// TIA Portal V20 export
// export: Created 2025-12-01T14:57:40.1723845Z, ExportSetting None, DisplayName Totally Integrated Automation Portal, DisplayVersion V20 Update 3, DisplayName TIA Portal Openness, DisplayVersion V20 Update 3, DisplayName TIA Portal Version Control Interface, DisplayVersion V20 Update 3, DisplayName STEP 7 Professional, DisplayVersion V20 Update 3, DisplayName STEP 7 Safety, DisplayVersion V20 Update 2, DisplayName WinCC Basic/Comfort/Advanced, DisplayVersion V20 Update 3, DisplayName WinCC Professional, DisplayVersion V20 Update 3, DisplayName WinCC Unified, DisplayVersion V20 Update 3
FUNCTION_BLOCK "FB159_M_PASO_E0E3_S0S3_RechazoFruta"   // FB159, LAD
TITLE = Control del Ramal de Salidas
{ S7_Optimized_Access := 'FALSE' }
AUTHOR : PASO
NAME : 20160509
VERSION : 3.3
// stored: AutoNumber false, SetENOAutomatically false
   VAR_INPUT
      Mesa : UInt;   // Mesa de la FB
      Error_Tx : Bool;   // Error en el Tx
      EnTension : Bool;   // Existe Tension en la Mesa
      Termico_Tx : Bool;   // Proteccion del Tx
      pHsMx_Carretilla : Bool;   // pHs de Carretilla
      pHsMx : Bool;   // pHs de la Mesa
      pHsMx_PR3 : Bool;   // pHs de Protrusion de la Mesa. Nota: No existe >> ON
      EnMovimiento_Tx : Bool;   // Avance o Retroceso del Tx
      MAnt_DescargaAct : Bool;   // E1 >> Mesa Anterior DescargaAct
      AVTF_MAnt_Mx : Bool;   // E1 >> Mesa Anterior AVTF
      P_Mens_MAnt_Mx : Bool;   // E1 >> Mesa Anterior P_Mens
      PTF_Mx_MSig : Bool;   // S3 >> Mesa Siguiente PTF
      FTF_Mx_MSig : Bool;   // S3 >> Mesa Siguiente FTF
      MSig_CargaAct : Bool;
      Mx_Centraje : Bool;   // Config >> Activar Centraje de Carga
      Mx_VelocidadLenta_In : Bool;   // Forzar a Velociada Lenta
      F_ENV_MENS_Mx : Bool;   // Fin de Envio de Mensaje
      OrdSal_S03 : Bool;   // Orden de Salida por S3
      OrdSal_S00 : Bool;   // Orden de Salida por S0
      V_CNT_pHsMx : Int := 1000;   // Valor de Presencia
      V_CNT_pHsMx_FTF : Int := 200;   // Valor para activar FTF. Nota: < = V_CNT_pHsMx.
      V_CNTSeg_pHsMx : Int := 2000;   // Valor de Seguriadad para Presencia
      V_CNT_PasoLenta : Int := 2000;   // Valor de Paso a Lenta
      V_CNT_AphsMx : Int := 500;   // Valor de Ausencia
      V_CNTSeg_ApHsMx : Int := 2000;   // Valor de Seguriadad para Ausencia
      V_TMP_Entrada : Int := 5000;   // Valor de Entrada de Carga >> E0
      V_TMP_Retirar : Int := 5000;   // Valor de Retirada de Carga >> S0
      V_CNT_Centrado : Int := 2000;   // Valor de Centrado de Carga
      V_CNT_Reposo : Int := 3000;   // Valor de Reposo de Carga Nota: > Centrado
      V_TOut_Tx_Mx : Int := 15000;   // TimeOut de Entrada por E1
      V_TMP_Protrusion : Int := 200;   // TMP de Protrusion
      V_CNT_PerdidapHs : Int := 1000;   // CNT de Perdida de pHs
   END_VAR
   VAR_OUTPUT
      P_EnvMens_PMx : Bool;   // Permiso de Enviar Mensaje de Presencia
      P_EnvMens_AMx : Bool;   // Permiso de Enviar Mensaje de Ausencia
      P_RecepOK_Mx : Bool;   // Recepcion OK
      PTF_MAnt_Mx : Bool;   // E1 >> Mesa Anterior PTF
      FTF_MAnt_Mx : Bool;   // E1 >> Mesa Anterior FTF
      AVTF_Mx_MSig : Bool;   // S3 >> Mesa Siguiente AVTF
      P_Mens_Mx_MSig : Bool;   // S3 >> Mesa Siguiente P_Mens
   END_VAR
   VAR
      Anular_prE1 : Bool;   // ???
      Anular_prS3 : Bool;   // ???
      Mx_ET00 : Bool;
      Mx_ET01 : Bool;
      Mx_ET02 : Bool;
      Mx_ET08 : Bool;
      Mx_ET09 : Bool;
      Mx_ET10 : Bool;
      Mx_ET11 : Bool;
      Mx_ET12 : Bool;
      Mx_ET110 : Bool;
      Mx_ET111 : Bool;
      Mx_ET40 : Bool;
      Mx_ET41 : Bool;
      Mx_ET42 : Bool;
      Mx_ET43 : Bool;
      Mx_ET140 : Bool;
      Mx_ET141 : Bool;
      Mx_ET50 : Bool;
      Mx_ET51 : Bool;
      Mx_ET150 : Bool;
      Mx_ET151 : Bool;
      Mx_ET90 : Bool;
      Mx_ET91 : Bool;
      Mx_ET190 : Bool;
      Mx_ET191 : Bool;
      Mx_ET192 : Bool;
      ProtocoloIniciado : Bool;   // Iniciado el Envio del Mensaje de Presencia
      CNT_pHsMx_FTF_OK : Bool;   // Enviar ya FTF
      CNT_pHsMx { S7_SetPoint := 'True'} : "FB910_CNT_UHS";   // CNT de la Presencia
      CNTSeg_pHsMx { S7_SetPoint := 'True'} : "FB910_CNT_UHS";   // CNT de Seguridad de la Presencia
      CNT_ApHsMx { S7_SetPoint := 'True'} : "FB910_CNT_UHS";   // CNT de la Ausencia
      CNTSeg_ApHsMx { S7_SetPoint := 'True'} : "FB910_CNT_UHS";   // CNT de Seguridad de la Ausencia
      TMP_Entrada { S7_SetPoint := 'True'} : "FB910_CNT_UHS";   // TMP de Entrada de Carga
      TMP_Retirar { S7_SetPoint := 'True'} : "FB910_CNT_UHS";   // TMP de Retirada de Carga
      CNT_Centrado { S7_SetPoint := 'True'} : "FB910_CNT_UHS";   // Contador de Centrado de Carga
      TMP_EnTension { S7_SetPoint := 'True'} : "FB910_CNT_UHS";
      TOut_Av_Mx { S7_SetPoint := 'True'} : "FB910_CNT_UHS";   // Time Out de Entrada de E1
      TMP_Protrusion { S7_SetPoint := 'True'} : "FB910_CNT_UHS";   // TMP de la Protrusion
      CNT_PerdidapHs { S7_SetPoint := 'True'} : "FB910_CNT_UHS";   // CNT de Perdida de pHs
      STAT_EnvMens_PMx : Bool;   // Interna >> Envio del Mensaje de Presencia
      STAT_EnvMens_AMx : Bool;   // Interna >> Envio de Mensaje de Ausencia
      STAT_FTF_MAnt_Mx : Bool;   // Interna >> FTF de MAnt >> Mx
      STAT_AVTF_Mx_MSig : Bool;   // Interna >> AVTF de Mx >> MSig
      MA_BalizaEntrada : Bool;   // ????
   END_VAR
   VAR_TEMP
      EstadoZona : "EstadoZona";   // Estado de Zona de la Mesa
      EstadoVI : "EstadosMesa";   // Estado del Vehiculo Inteliguente de la Mesa
      ConfigFB : "UDT_ConfigFB";   // Configuracion de la FB de la Mesa
      V_Protrusion : Int;
      Aux_ET00 : Bool;
   END_VAR
BEGIN

REGION Network 1: INICIALIZAR - Recoger las Variables de Estado de la Mesa
   // Se recoge - Estado_CBx
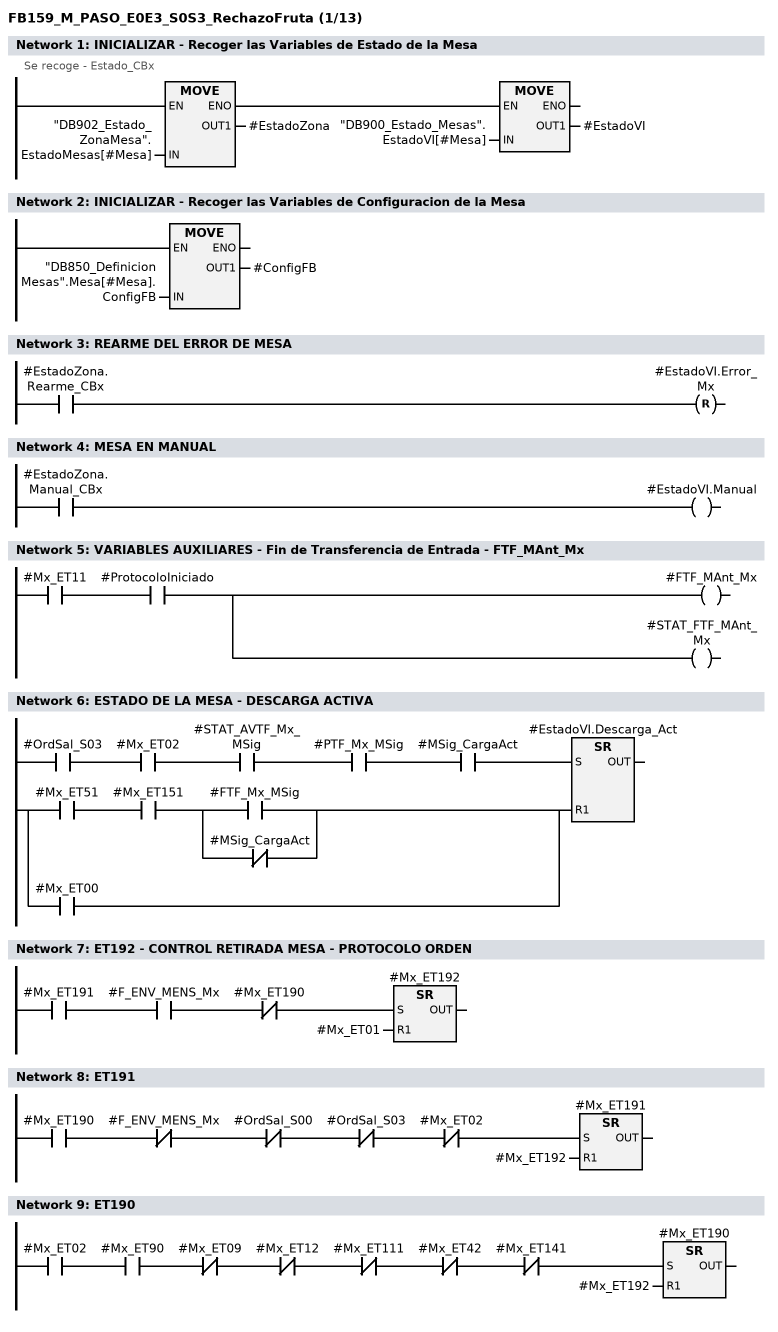
   RUNG wire#powerrail
      Move(in := "DB902_Estado_ZonaMesa".EstadoMesas[#Mesa], out1 => #EstadoZona)
      Move(in := "DB900_Estado_Mesas".EstadoVI[#Mesa], out1 => #EstadoVI)
   END_RUNG
   // the same network as SCL:
   #EstadoZona := "DB902_Estado_ZonaMesa".EstadoMesas[#Mesa];
   #EstadoVI := "DB900_Estado_Mesas".EstadoVI[#Mesa];
END_REGION

REGION Network 2: INICIALIZAR - Recoger las Variables de Configuracion de la Mesa
   RUNG wire#powerrail
      Move(in := "DB850_DefinicionMesas".Mesa[#Mesa].ConfigFB, out1 => #ConfigFB)
   END_RUNG
   // the same network as SCL:
   #ConfigFB := "DB850_DefinicionMesas".Mesa[#Mesa].ConfigFB;
END_REGION

REGION Network 3: REARME DEL ERROR DE MESA
   RUNG wire#powerrail
      Contact( #EstadoZona.Rearme_CBx )
      R_Coil( #EstadoVI.Error_Mx )
   END_RUNG
   // the same network as SCL:
   IF #EstadoZona.Rearme_CBx THEN #EstadoVI.Error_Mx := FALSE; END_IF;
END_REGION

REGION Network 4: MESA EN MANUAL
   RUNG wire#powerrail
      Contact( #EstadoZona.Manual_CBx )
      Coil( #EstadoVI.Manual )
   END_RUNG
   // the same network as SCL:
   #EstadoVI.Manual := #EstadoZona.Manual_CBx;
END_REGION

REGION Network 5: VARIABLES AUXILIARES - Fin de Transferencia de Entrada - FTF_MAnt_Mx
   RUNG wire#powerrail
      Contact( #Mx_ET11 )
      Contact( #ProtocoloIniciado )
      wire#w1
      Coil( #FTF_MAnt_Mx )
   END_RUNG
   RUNG wire#w1
      Coil( #STAT_FTF_MAnt_Mx )
   END_RUNG
   // the same network as SCL:
   #FTF_MAnt_Mx := #Mx_ET11 AND #ProtocoloIniciado;
   #STAT_FTF_MAnt_Mx := #FTF_MAnt_Mx;
END_REGION

REGION Network 6: ESTADO DE LA MESA - DESCARGA ACTIVA
   RUNG wire#powerrail
      Contact( #OrdSal_S03 )
      Contact( #Mx_ET02 )
      Contact( #STAT_AVTF_Mx_MSig )
      Contact( #PTF_Mx_MSig )
      Contact( #MSig_CargaAct )
      S_SR(operand := #EstadoVI.Descarga_Act, r1 := wire#w2)
   END_RUNG
   RUNG wire#powerrail
      Contact( #Mx_ET51 )
      Contact( #Mx_ET151 )
      wire#w1
      Contact( #FTF_Mx_MSig )
   END_RUNG wire#w2
   RUNG wire#w1
      I_Contact( #MSig_CargaAct )
   END_RUNG wire#w2
   RUNG wire#powerrail
      Contact( #Mx_ET00 )
   END_RUNG wire#w2
   // the same network as SCL:
   IF #OrdSal_S03 AND #Mx_ET02 AND #STAT_AVTF_Mx_MSig AND #PTF_Mx_MSig AND #MSig_CargaAct THEN
       #EstadoVI.Descarga_Act := TRUE;   // SR flip-flop
   END_IF;
   IF (#Mx_ET51 AND #Mx_ET151 AND (#FTF_Mx_MSig OR NOT #MSig_CargaAct)) OR #Mx_ET00 THEN
       #EstadoVI.Descarga_Act := FALSE;
   END_IF;
END_REGION

REGION Network 7: ET192 - CONTROL RETIRADA MESA - PROTOCOLO ORDEN
   RUNG wire#powerrail
      Contact( #Mx_ET191 )
      Contact( #F_ENV_MENS_Mx )
      I_Contact( #Mx_ET190 )
      S_SR(operand := #Mx_ET192, r1 := #Mx_ET01)
   END_RUNG
   // the same network as SCL:
   IF #Mx_ET191 AND #F_ENV_MENS_Mx AND NOT #Mx_ET190 THEN
       #Mx_ET192 := TRUE;   // SR flip-flop
   END_IF;
   IF #Mx_ET01 THEN #Mx_ET192 := FALSE; END_IF;
END_REGION

REGION Network 8: ET191
   RUNG wire#powerrail
      Contact( #Mx_ET190 )
      I_Contact( #F_ENV_MENS_Mx )
      I_Contact( #OrdSal_S00 )
      I_Contact( #OrdSal_S03 )
      I_Contact( #Mx_ET02 )
      S_SR(operand := #Mx_ET191, r1 := #Mx_ET192)
   END_RUNG
   // the same network as SCL:
   IF #Mx_ET190 AND NOT #F_ENV_MENS_Mx AND NOT #OrdSal_S00 AND NOT #OrdSal_S03 AND NOT #Mx_ET02 THEN
       #Mx_ET191 := TRUE;   // SR flip-flop
   END_IF;
   IF #Mx_ET192 THEN #Mx_ET191 := FALSE; END_IF;
END_REGION

REGION Network 9: ET190
   RUNG wire#powerrail
      Contact( #Mx_ET02 )
      Contact( #Mx_ET90 )
      I_Contact( #Mx_ET09 )
      I_Contact( #Mx_ET12 )
      I_Contact( #Mx_ET111 )
      I_Contact( #Mx_ET42 )
      I_Contact( #Mx_ET141 )
      S_SR(operand := #Mx_ET190, r1 := #Mx_ET192)
   END_RUNG
   // the same network as SCL:
   IF #Mx_ET02 AND #Mx_ET90 AND NOT #Mx_ET09 AND NOT #Mx_ET12 AND NOT #Mx_ET111 AND NOT #Mx_ET42 AND NOT #Mx_ET141 THEN
       #Mx_ET190 := TRUE;   // SR flip-flop
   END_IF;
   IF #Mx_ET192 THEN #Mx_ET190 := FALSE; END_IF;
END_REGION

REGION Network 10: ET91 - CONTROL RETIRAR DE MESA
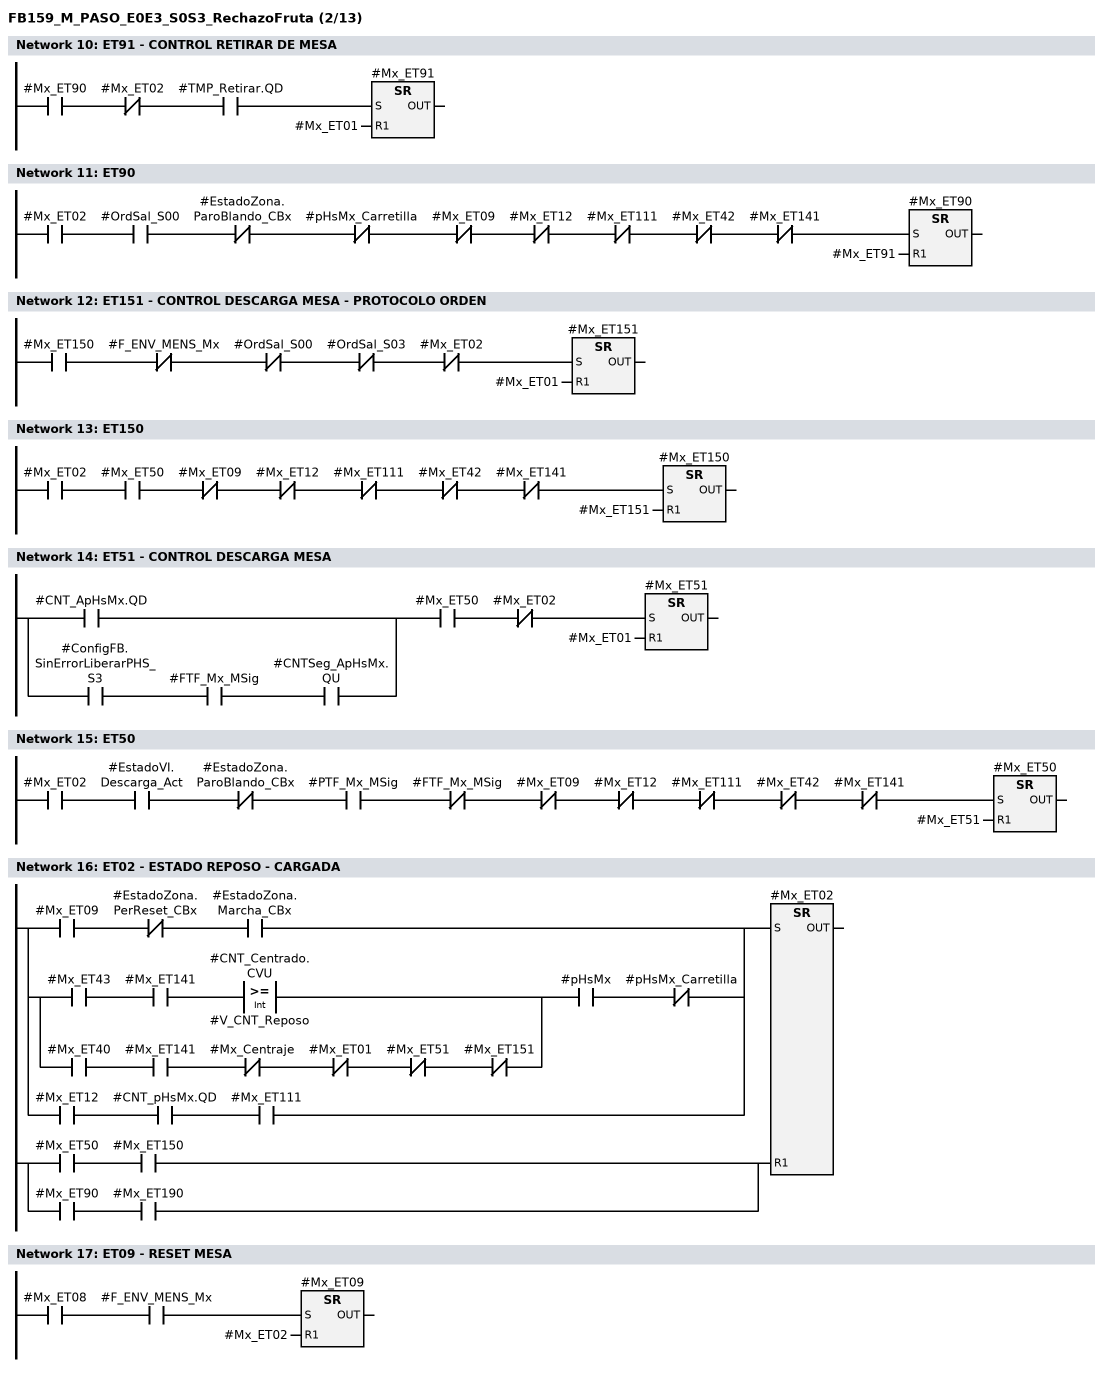
   RUNG wire#powerrail
      Contact( #Mx_ET90 )
      I_Contact( #Mx_ET02 )
      Contact( #TMP_Retirar.QD )
      S_SR(operand := #Mx_ET91, r1 := #Mx_ET01)
   END_RUNG
   // the same network as SCL:
   IF #Mx_ET90 AND NOT #Mx_ET02 AND #TMP_Retirar.QD THEN
       #Mx_ET91 := TRUE;   // SR flip-flop
   END_IF;
   IF #Mx_ET01 THEN #Mx_ET91 := FALSE; END_IF;
END_REGION

REGION Network 11: ET90
   RUNG wire#powerrail
      Contact( #Mx_ET02 )
      Contact( #OrdSal_S00 )
      I_Contact( #EstadoZona.ParoBlando_CBx )
      I_Contact( #pHsMx_Carretilla )
      I_Contact( #Mx_ET09 )
      I_Contact( #Mx_ET12 )
      I_Contact( #Mx_ET111 )
      I_Contact( #Mx_ET42 )
      I_Contact( #Mx_ET141 )
      S_SR(operand := #Mx_ET90, r1 := #Mx_ET91)
   END_RUNG
   // the same network as SCL:
   IF #Mx_ET02 AND #OrdSal_S00 AND NOT #EstadoZona.ParoBlando_CBx AND NOT #pHsMx_Carretilla AND NOT #Mx_ET09 AND NOT #Mx_ET12 AND NOT #Mx_ET111 AND NOT #Mx_ET42 AND NOT #Mx_ET141 THEN
       #Mx_ET90 := TRUE;   // SR flip-flop
   END_IF;
   IF #Mx_ET91 THEN #Mx_ET90 := FALSE; END_IF;
END_REGION

REGION Network 12: ET151 - CONTROL DESCARGA MESA - PROTOCOLO ORDEN
   RUNG wire#powerrail
      Contact( #Mx_ET150 )
      I_Contact( #F_ENV_MENS_Mx )
      I_Contact( #OrdSal_S00 )
      I_Contact( #OrdSal_S03 )
      I_Contact( #Mx_ET02 )
      S_SR(operand := #Mx_ET151, r1 := #Mx_ET01)
   END_RUNG
   // the same network as SCL:
   IF #Mx_ET150 AND NOT #F_ENV_MENS_Mx AND NOT #OrdSal_S00 AND NOT #OrdSal_S03 AND NOT #Mx_ET02 THEN
       #Mx_ET151 := TRUE;   // SR flip-flop
   END_IF;
   IF #Mx_ET01 THEN #Mx_ET151 := FALSE; END_IF;
END_REGION

REGION Network 13: ET150
   RUNG wire#powerrail
      Contact( #Mx_ET02 )
      Contact( #Mx_ET50 )
      I_Contact( #Mx_ET09 )
      I_Contact( #Mx_ET12 )
      I_Contact( #Mx_ET111 )
      I_Contact( #Mx_ET42 )
      I_Contact( #Mx_ET141 )
      S_SR(operand := #Mx_ET150, r1 := #Mx_ET151)
   END_RUNG
   // the same network as SCL:
   IF #Mx_ET02 AND #Mx_ET50 AND NOT #Mx_ET09 AND NOT #Mx_ET12 AND NOT #Mx_ET111 AND NOT #Mx_ET42 AND NOT #Mx_ET141 THEN
       #Mx_ET150 := TRUE;   // SR flip-flop
   END_IF;
   IF #Mx_ET151 THEN #Mx_ET150 := FALSE; END_IF;
END_REGION

REGION Network 14: ET51 - CONTROL DESCARGA MESA
   RUNG wire#powerrail
      Contact( #CNT_ApHsMx.QD )
      wire#w1
      Contact( #Mx_ET50 )
      I_Contact( #Mx_ET02 )
      S_SR(operand := #Mx_ET51, r1 := #Mx_ET01)
   END_RUNG
   RUNG wire#powerrail
      Contact( #ConfigFB.SinErrorLiberarPHS_S3 )
      Contact( #FTF_Mx_MSig )
      Contact( #CNTSeg_ApHsMx.QU )
   END_RUNG wire#w1
   // the same network as SCL:
   IF (#CNT_ApHsMx.QD OR (#ConfigFB.SinErrorLiberarPHS_S3 AND #FTF_Mx_MSig AND #CNTSeg_ApHsMx.QU)) AND #Mx_ET50 AND NOT #Mx_ET02 THEN
       #Mx_ET51 := TRUE;   // SR flip-flop
   END_IF;
   IF #Mx_ET01 THEN #Mx_ET51 := FALSE; END_IF;
END_REGION

REGION Network 15: ET50
   RUNG wire#powerrail
      Contact( #Mx_ET02 )
      Contact( #EstadoVI.Descarga_Act )
      I_Contact( #EstadoZona.ParoBlando_CBx )
      Contact( #PTF_Mx_MSig )
      I_Contact( #FTF_Mx_MSig )
      I_Contact( #Mx_ET09 )
      I_Contact( #Mx_ET12 )
      I_Contact( #Mx_ET111 )
      I_Contact( #Mx_ET42 )
      I_Contact( #Mx_ET141 )
      S_SR(operand := #Mx_ET50, r1 := #Mx_ET51)
   END_RUNG
   // the same network as SCL:
   IF #Mx_ET02 AND #EstadoVI.Descarga_Act AND NOT #EstadoZona.ParoBlando_CBx AND #PTF_Mx_MSig AND NOT #FTF_Mx_MSig AND NOT #Mx_ET09 AND NOT #Mx_ET12 AND NOT #Mx_ET111 AND NOT #Mx_ET42 AND NOT #Mx_ET141 THEN
       #Mx_ET50 := TRUE;   // SR flip-flop
   END_IF;
   IF #Mx_ET51 THEN #Mx_ET50 := FALSE; END_IF;
END_REGION

REGION Network 16: ET02 - ESTADO REPOSO - CARGADA
   RUNG wire#powerrail
      Contact( #Mx_ET09 )
      I_Contact( #EstadoZona.PerReset_CBx )
      Contact( #EstadoZona.Marcha_CBx )
      wire#w1
      S_SR(operand := #Mx_ET02, r1 := wire#w3)
   END_RUNG
   RUNG wire#powerrail
      Contact( #Mx_ET43 )
      Contact( #Mx_ET141 )
      { S7_Templates := "SrcType := Int" } GE_Contact(in1 := #CNT_Centrado.CVU, in2 := #V_CNT_Reposo)
      wire#w2
      Contact( #pHsMx )
      I_Contact( #pHsMx_Carretilla )
   END_RUNG wire#w1
   RUNG wire#powerrail
      Contact( #Mx_ET40 )
      Contact( #Mx_ET141 )
      I_Contact( #Mx_Centraje )
      I_Contact( #Mx_ET01 )
      I_Contact( #Mx_ET51 )
      I_Contact( #Mx_ET151 )
   END_RUNG wire#w2
   RUNG wire#powerrail
      Contact( #Mx_ET12 )
      Contact( #CNT_pHsMx.QD )
      Contact( #Mx_ET111 )
   END_RUNG wire#w1
   RUNG wire#powerrail
      Contact( #Mx_ET50 )
      Contact( #Mx_ET150 )
   END_RUNG wire#w3
   RUNG wire#powerrail
      Contact( #Mx_ET90 )
      Contact( #Mx_ET190 )
   END_RUNG wire#w3
   // the same network as SCL:
   IF (#Mx_ET09 AND NOT #EstadoZona.PerReset_CBx AND #EstadoZona.Marcha_CBx) OR (((#Mx_ET43 AND #Mx_ET141 AND (#CNT_Centrado.CVU >= #V_CNT_Reposo)) OR (#Mx_ET40 AND #Mx_ET141 AND NOT #Mx_Centraje AND NOT #Mx_ET01 AND NOT #Mx_ET51 AND NOT #Mx_ET151)) AND #pHsMx AND NOT #pHsMx_Carretilla) OR (#Mx_ET12 AND #CNT_pHsMx.QD AND #Mx_ET111) THEN
       #Mx_ET02 := TRUE;   // SR flip-flop
   END_IF;
   IF (#Mx_ET50 AND #Mx_ET150) OR (#Mx_ET90 AND #Mx_ET190) THEN #Mx_ET02 := FALSE; END_IF;
END_REGION

REGION Network 17: ET09 - RESET MESA
   RUNG wire#powerrail
      Contact( #Mx_ET08 )
      Contact( #F_ENV_MENS_Mx )
      S_SR(operand := #Mx_ET09, r1 := #Mx_ET02)
   END_RUNG
   // the same network as SCL:
   IF #Mx_ET08 AND #F_ENV_MENS_Mx THEN
       #Mx_ET09 := TRUE;   // SR flip-flop
   END_IF;
   IF #Mx_ET02 THEN #Mx_ET09 := FALSE; END_IF;
END_REGION

REGION Network 18: ET08
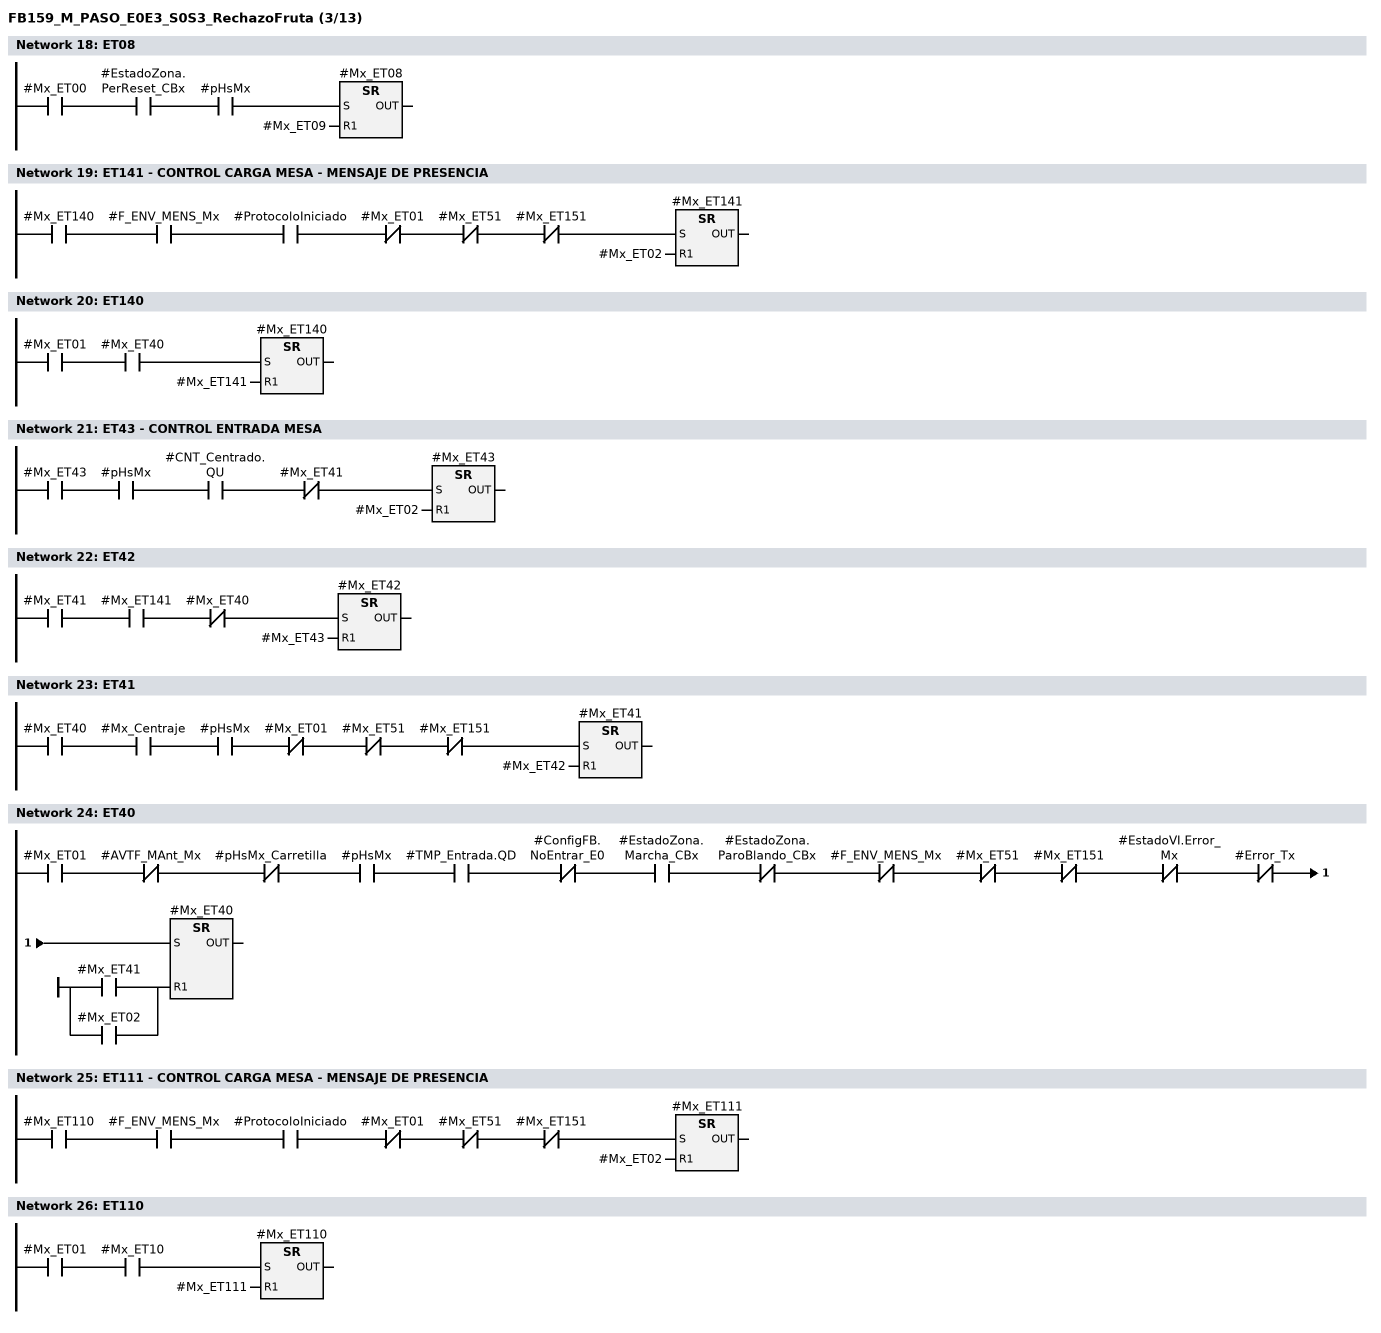
   RUNG wire#powerrail
      Contact( #Mx_ET00 )
      Contact( #EstadoZona.PerReset_CBx )
      Contact( #pHsMx )
      S_SR(operand := #Mx_ET08, r1 := #Mx_ET09)
   END_RUNG
   // the same network as SCL:
   IF #Mx_ET00 AND #EstadoZona.PerReset_CBx AND #pHsMx THEN
       #Mx_ET08 := TRUE;   // SR flip-flop
   END_IF;
   IF #Mx_ET09 THEN #Mx_ET08 := FALSE; END_IF;
END_REGION

REGION Network 19: ET141 - CONTROL CARGA MESA - MENSAJE DE PRESENCIA
   RUNG wire#powerrail
      Contact( #Mx_ET140 )
      Contact( #F_ENV_MENS_Mx )
      Contact( #ProtocoloIniciado )
      I_Contact( #Mx_ET01 )
      I_Contact( #Mx_ET51 )
      I_Contact( #Mx_ET151 )
      S_SR(operand := #Mx_ET141, r1 := #Mx_ET02)
   END_RUNG
   // the same network as SCL:
   IF #Mx_ET140 AND #F_ENV_MENS_Mx AND #ProtocoloIniciado AND NOT #Mx_ET01 AND NOT #Mx_ET51 AND NOT #Mx_ET151 THEN
       #Mx_ET141 := TRUE;   // SR flip-flop
   END_IF;
   IF #Mx_ET02 THEN #Mx_ET141 := FALSE; END_IF;
END_REGION

REGION Network 20: ET140
   RUNG wire#powerrail
      Contact( #Mx_ET01 )
      Contact( #Mx_ET40 )
      S_SR(operand := #Mx_ET140, r1 := #Mx_ET141)
   END_RUNG
   // the same network as SCL:
   IF #Mx_ET01 AND #Mx_ET40 THEN
       #Mx_ET140 := TRUE;   // SR flip-flop
   END_IF;
   IF #Mx_ET141 THEN #Mx_ET140 := FALSE; END_IF;
END_REGION

REGION Network 21: ET43 - CONTROL ENTRADA MESA
   RUNG wire#powerrail
      Contact( #Mx_ET43 )
      Contact( #pHsMx )
      Contact( #CNT_Centrado.QU )
      I_Contact( #Mx_ET41 )
      S_SR(operand := #Mx_ET43, r1 := #Mx_ET02)
   END_RUNG
   // the same network as SCL:
   IF #Mx_ET43 AND #pHsMx AND #CNT_Centrado.QU AND NOT #Mx_ET41 THEN
       #Mx_ET43 := TRUE;   // SR flip-flop
   END_IF;
   IF #Mx_ET02 THEN #Mx_ET43 := FALSE; END_IF;
END_REGION

REGION Network 22: ET42
   RUNG wire#powerrail
      Contact( #Mx_ET41 )
      Contact( #Mx_ET141 )
      I_Contact( #Mx_ET40 )
      S_SR(operand := #Mx_ET42, r1 := #Mx_ET43)
   END_RUNG
   // the same network as SCL:
   IF #Mx_ET41 AND #Mx_ET141 AND NOT #Mx_ET40 THEN
       #Mx_ET42 := TRUE;   // SR flip-flop
   END_IF;
   IF #Mx_ET43 THEN #Mx_ET42 := FALSE; END_IF;
END_REGION

REGION Network 23: ET41
   RUNG wire#powerrail
      Contact( #Mx_ET40 )
      Contact( #Mx_Centraje )
      Contact( #pHsMx )
      I_Contact( #Mx_ET01 )
      I_Contact( #Mx_ET51 )
      I_Contact( #Mx_ET151 )
      S_SR(operand := #Mx_ET41, r1 := #Mx_ET42)
   END_RUNG
   // the same network as SCL:
   IF #Mx_ET40 AND #Mx_Centraje AND #pHsMx AND NOT #Mx_ET01 AND NOT #Mx_ET51 AND NOT #Mx_ET151 THEN
       #Mx_ET41 := TRUE;   // SR flip-flop
   END_IF;
   IF #Mx_ET42 THEN #Mx_ET41 := FALSE; END_IF;
END_REGION

REGION Network 24: ET40
   RUNG wire#powerrail
      Contact( #Mx_ET01 )
      I_Contact( #AVTF_MAnt_Mx )
      I_Contact( #pHsMx_Carretilla )
      Contact( #pHsMx )
      Contact( #TMP_Entrada.QD )
      I_Contact( #ConfigFB.NoEntrar_E0 )
      Contact( #EstadoZona.Marcha_CBx )
      I_Contact( #EstadoZona.ParoBlando_CBx )
      I_Contact( #F_ENV_MENS_Mx )
      I_Contact( #Mx_ET51 )
      I_Contact( #Mx_ET151 )
      I_Contact( #EstadoVI.Error_Mx )
      I_Contact( #Error_Tx )
      S_SR(operand := #Mx_ET40, r1 := wire#w1)
   END_RUNG
   RUNG wire#powerrail
      Contact( #Mx_ET41 )
   END_RUNG wire#w1
   RUNG wire#powerrail
      Contact( #Mx_ET02 )
   END_RUNG wire#w1
   // the same network as SCL:
   IF #Mx_ET01 AND NOT #AVTF_MAnt_Mx AND NOT #pHsMx_Carretilla AND #pHsMx AND #TMP_Entrada.QD AND NOT #ConfigFB.NoEntrar_E0 AND #EstadoZona.Marcha_CBx AND NOT #EstadoZona.ParoBlando_CBx AND NOT #F_ENV_MENS_Mx AND NOT #Mx_ET51 AND NOT #Mx_ET151 AND NOT #EstadoVI.Error_Mx AND NOT #Error_Tx THEN
       #Mx_ET40 := TRUE;   // SR flip-flop
   END_IF;
   IF #Mx_ET41 OR #Mx_ET02 THEN #Mx_ET40 := FALSE; END_IF;
END_REGION

REGION Network 25: ET111 - CONTROL CARGA MESA - MENSAJE DE PRESENCIA
   RUNG wire#powerrail
      Contact( #Mx_ET110 )
      Contact( #F_ENV_MENS_Mx )
      Contact( #ProtocoloIniciado )
      I_Contact( #Mx_ET01 )
      I_Contact( #Mx_ET51 )
      I_Contact( #Mx_ET151 )
      S_SR(operand := #Mx_ET111, r1 := #Mx_ET02)
   END_RUNG
   // the same network as SCL:
   IF #Mx_ET110 AND #F_ENV_MENS_Mx AND #ProtocoloIniciado AND NOT #Mx_ET01 AND NOT #Mx_ET51 AND NOT #Mx_ET151 THEN
       #Mx_ET111 := TRUE;   // SR flip-flop
   END_IF;
   IF #Mx_ET02 THEN #Mx_ET111 := FALSE; END_IF;
END_REGION

REGION Network 26: ET110
   RUNG wire#powerrail
      Contact( #Mx_ET01 )
      Contact( #Mx_ET10 )
      S_SR(operand := #Mx_ET110, r1 := #Mx_ET111)
   END_RUNG
   // the same network as SCL:
   IF #Mx_ET01 AND #Mx_ET10 THEN
       #Mx_ET110 := TRUE;   // SR flip-flop
   END_IF;
   IF #Mx_ET111 THEN #Mx_ET110 := FALSE; END_IF;
END_REGION

REGION Network 27: ET12 - CONTROL CARGA MESA
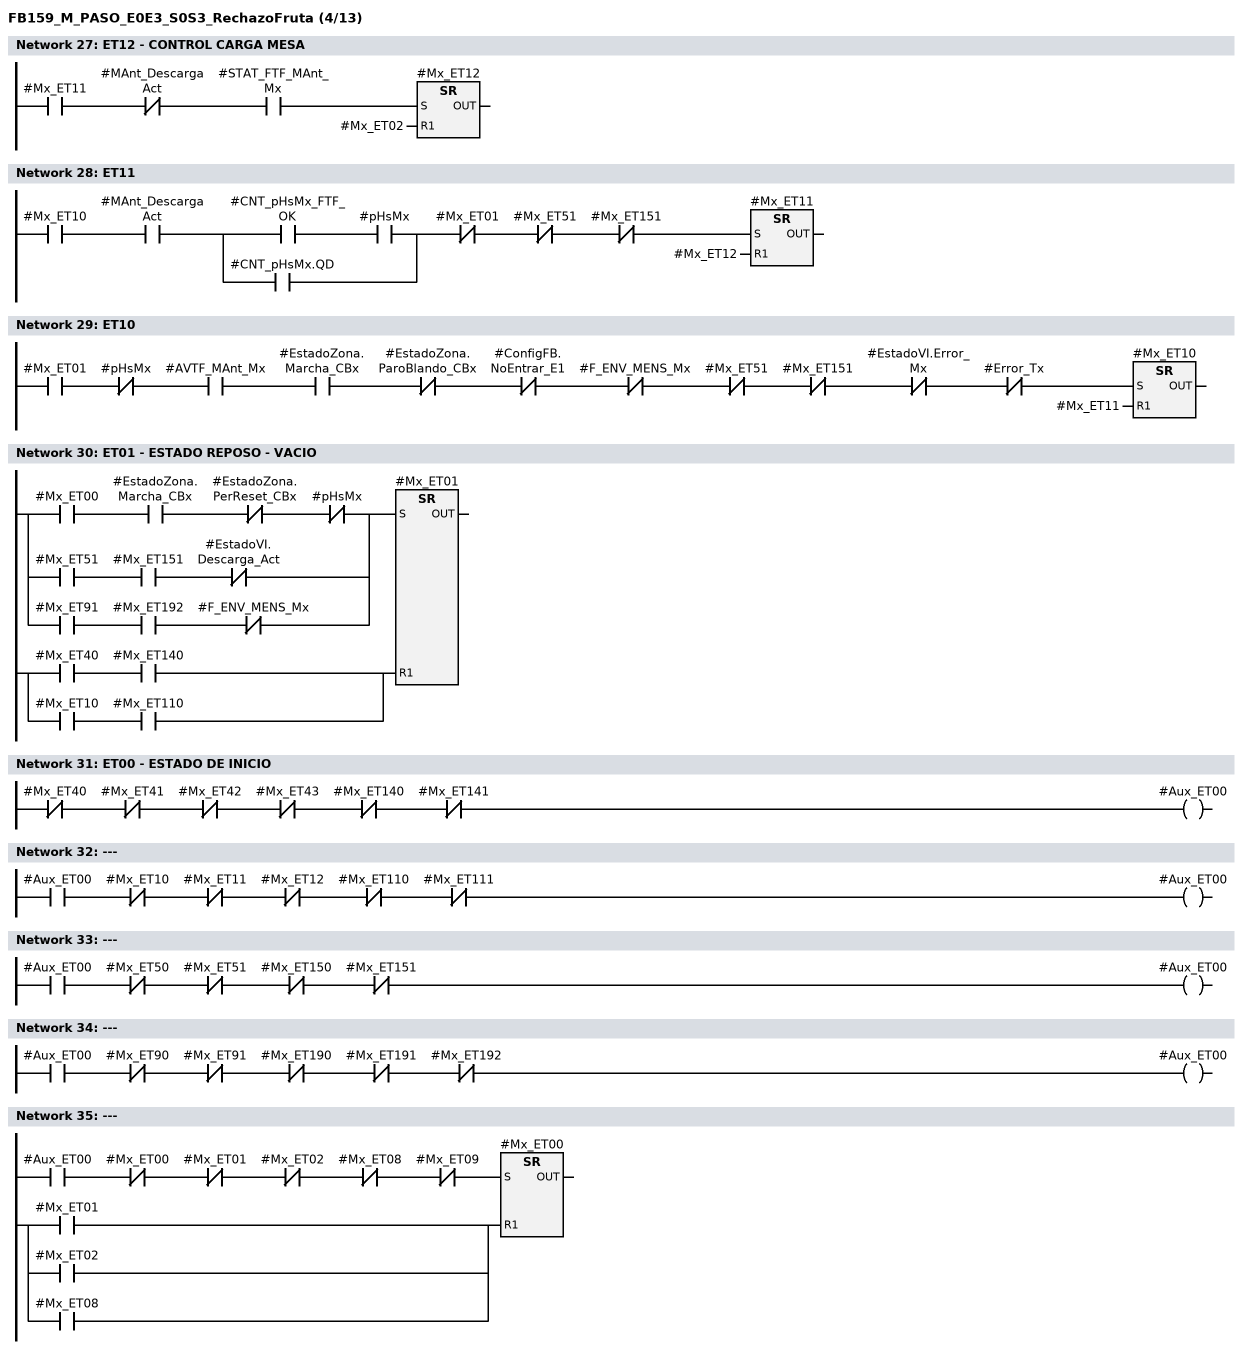
   RUNG wire#powerrail
      Contact( #Mx_ET11 )
      I_Contact( #MAnt_DescargaAct )
      Contact( #STAT_FTF_MAnt_Mx )
      S_SR(operand := #Mx_ET12, r1 := #Mx_ET02)
   END_RUNG
   // the same network as SCL:
   IF #Mx_ET11 AND NOT #MAnt_DescargaAct AND #STAT_FTF_MAnt_Mx THEN
       #Mx_ET12 := TRUE;   // SR flip-flop
   END_IF;
   IF #Mx_ET02 THEN #Mx_ET12 := FALSE; END_IF;
END_REGION

REGION Network 28: ET11
   RUNG wire#powerrail
      Contact( #Mx_ET10 )
      Contact( #MAnt_DescargaAct )
      wire#w1
      Contact( #CNT_pHsMx_FTF_OK )
      Contact( #pHsMx )
      wire#w2
      I_Contact( #Mx_ET01 )
      I_Contact( #Mx_ET51 )
      I_Contact( #Mx_ET151 )
      S_SR(operand := #Mx_ET11, r1 := #Mx_ET12)
   END_RUNG
   RUNG wire#w1
      Contact( #CNT_pHsMx.QD )
   END_RUNG wire#w2
   // the same network as SCL:
   IF #Mx_ET10 AND #MAnt_DescargaAct AND ((#CNT_pHsMx_FTF_OK AND #pHsMx) OR #CNT_pHsMx.QD) AND NOT #Mx_ET01 AND NOT #Mx_ET51 AND NOT #Mx_ET151 THEN
       #Mx_ET11 := TRUE;   // SR flip-flop
   END_IF;
   IF #Mx_ET12 THEN #Mx_ET11 := FALSE; END_IF;
END_REGION

REGION Network 29: ET10
   RUNG wire#powerrail
      Contact( #Mx_ET01 )
      I_Contact( #pHsMx )
      Contact( #AVTF_MAnt_Mx )
      Contact( #EstadoZona.Marcha_CBx )
      I_Contact( #EstadoZona.ParoBlando_CBx )
      I_Contact( #ConfigFB.NoEntrar_E1 )
      I_Contact( #F_ENV_MENS_Mx )
      I_Contact( #Mx_ET51 )
      I_Contact( #Mx_ET151 )
      I_Contact( #EstadoVI.Error_Mx )
      I_Contact( #Error_Tx )
      S_SR(operand := #Mx_ET10, r1 := #Mx_ET11)
   END_RUNG
   // the same network as SCL:
   IF #Mx_ET01 AND NOT #pHsMx AND #AVTF_MAnt_Mx AND #EstadoZona.Marcha_CBx AND NOT #EstadoZona.ParoBlando_CBx AND NOT #ConfigFB.NoEntrar_E1 AND NOT #F_ENV_MENS_Mx AND NOT #Mx_ET51 AND NOT #Mx_ET151 AND NOT #EstadoVI.Error_Mx AND NOT #Error_Tx THEN
       #Mx_ET10 := TRUE;   // SR flip-flop
   END_IF;
   IF #Mx_ET11 THEN #Mx_ET10 := FALSE; END_IF;
END_REGION

REGION Network 30: ET01 - ESTADO REPOSO - VACIO
   RUNG wire#powerrail
      Contact( #Mx_ET00 )
      Contact( #EstadoZona.Marcha_CBx )
      I_Contact( #EstadoZona.PerReset_CBx )
      I_Contact( #pHsMx )
      wire#w1
      S_SR(operand := #Mx_ET01, r1 := wire#w2)
   END_RUNG
   RUNG wire#powerrail
      Contact( #Mx_ET51 )
      Contact( #Mx_ET151 )
      I_Contact( #EstadoVI.Descarga_Act )
   END_RUNG wire#w1
   RUNG wire#powerrail
      Contact( #Mx_ET91 )
      Contact( #Mx_ET192 )
      I_Contact( #F_ENV_MENS_Mx )
   END_RUNG wire#w1
   RUNG wire#powerrail
      Contact( #Mx_ET40 )
      Contact( #Mx_ET140 )
   END_RUNG wire#w2
   RUNG wire#powerrail
      Contact( #Mx_ET10 )
      Contact( #Mx_ET110 )
   END_RUNG wire#w2
   // the same network as SCL:
   IF (#Mx_ET00 AND #EstadoZona.Marcha_CBx AND NOT #EstadoZona.PerReset_CBx AND NOT #pHsMx) OR (#Mx_ET51 AND #Mx_ET151 AND NOT #EstadoVI.Descarga_Act) OR (#Mx_ET91 AND #Mx_ET192 AND NOT #F_ENV_MENS_Mx) THEN
       #Mx_ET01 := TRUE;   // SR flip-flop
   END_IF;
   IF (#Mx_ET40 AND #Mx_ET140) OR (#Mx_ET10 AND #Mx_ET110) THEN #Mx_ET01 := FALSE; END_IF;
END_REGION

REGION Network 31: ET00 - ESTADO DE INICIO
   RUNG wire#powerrail
      I_Contact( #Mx_ET40 )
      I_Contact( #Mx_ET41 )
      I_Contact( #Mx_ET42 )
      I_Contact( #Mx_ET43 )
      I_Contact( #Mx_ET140 )
      I_Contact( #Mx_ET141 )
      Coil( #Aux_ET00 )
   END_RUNG
   // the same network as SCL:
   #Aux_ET00 := NOT #Mx_ET40 AND NOT #Mx_ET41 AND NOT #Mx_ET42 AND NOT #Mx_ET43 AND NOT #Mx_ET140 AND NOT #Mx_ET141;
END_REGION

REGION Network 32: ---
   RUNG wire#powerrail
      Contact( #Aux_ET00 )
      I_Contact( #Mx_ET10 )
      I_Contact( #Mx_ET11 )
      I_Contact( #Mx_ET12 )
      I_Contact( #Mx_ET110 )
      I_Contact( #Mx_ET111 )
      Coil( #Aux_ET00 )
   END_RUNG
   // the same network as SCL:
   #Aux_ET00 := #Aux_ET00 AND NOT #Mx_ET10 AND NOT #Mx_ET11 AND NOT #Mx_ET12 AND NOT #Mx_ET110 AND NOT #Mx_ET111;
END_REGION

REGION Network 33: ---
   RUNG wire#powerrail
      Contact( #Aux_ET00 )
      I_Contact( #Mx_ET50 )
      I_Contact( #Mx_ET51 )
      I_Contact( #Mx_ET150 )
      I_Contact( #Mx_ET151 )
      Coil( #Aux_ET00 )
   END_RUNG
   // the same network as SCL:
   #Aux_ET00 := #Aux_ET00 AND NOT #Mx_ET50 AND NOT #Mx_ET51 AND NOT #Mx_ET150 AND NOT #Mx_ET151;
END_REGION

REGION Network 34: ---
   RUNG wire#powerrail
      Contact( #Aux_ET00 )
      I_Contact( #Mx_ET90 )
      I_Contact( #Mx_ET91 )
      I_Contact( #Mx_ET190 )
      I_Contact( #Mx_ET191 )
      I_Contact( #Mx_ET192 )
      Coil( #Aux_ET00 )
   END_RUNG
   // the same network as SCL:
   #Aux_ET00 := #Aux_ET00 AND NOT #Mx_ET90 AND NOT #Mx_ET91 AND NOT #Mx_ET190 AND NOT #Mx_ET191 AND NOT #Mx_ET192;
END_REGION

REGION Network 35: ---
   RUNG wire#powerrail
      Contact( #Aux_ET00 )
      I_Contact( #Mx_ET00 )
      I_Contact( #Mx_ET01 )
      I_Contact( #Mx_ET02 )
      I_Contact( #Mx_ET08 )
      I_Contact( #Mx_ET09 )
      S_SR(operand := #Mx_ET00, r1 := wire#w1)
   END_RUNG
   RUNG wire#powerrail
      Contact( #Mx_ET01 )
   END_RUNG wire#w1
   RUNG wire#powerrail
      Contact( #Mx_ET02 )
   END_RUNG wire#w1
   RUNG wire#powerrail
      Contact( #Mx_ET08 )
   END_RUNG wire#w1
   // the same network as SCL:
   IF #Aux_ET00 AND NOT #Mx_ET00 AND NOT #Mx_ET01 AND NOT #Mx_ET02 AND NOT #Mx_ET08 AND NOT #Mx_ET09 THEN
       #Mx_ET00 := TRUE;   // SR flip-flop
   END_IF;
   IF #Mx_ET01 OR #Mx_ET02 OR #Mx_ET08 THEN #Mx_ET00 := FALSE; END_IF;
END_REGION

REGION Network 36: TMP - Espera En Tension
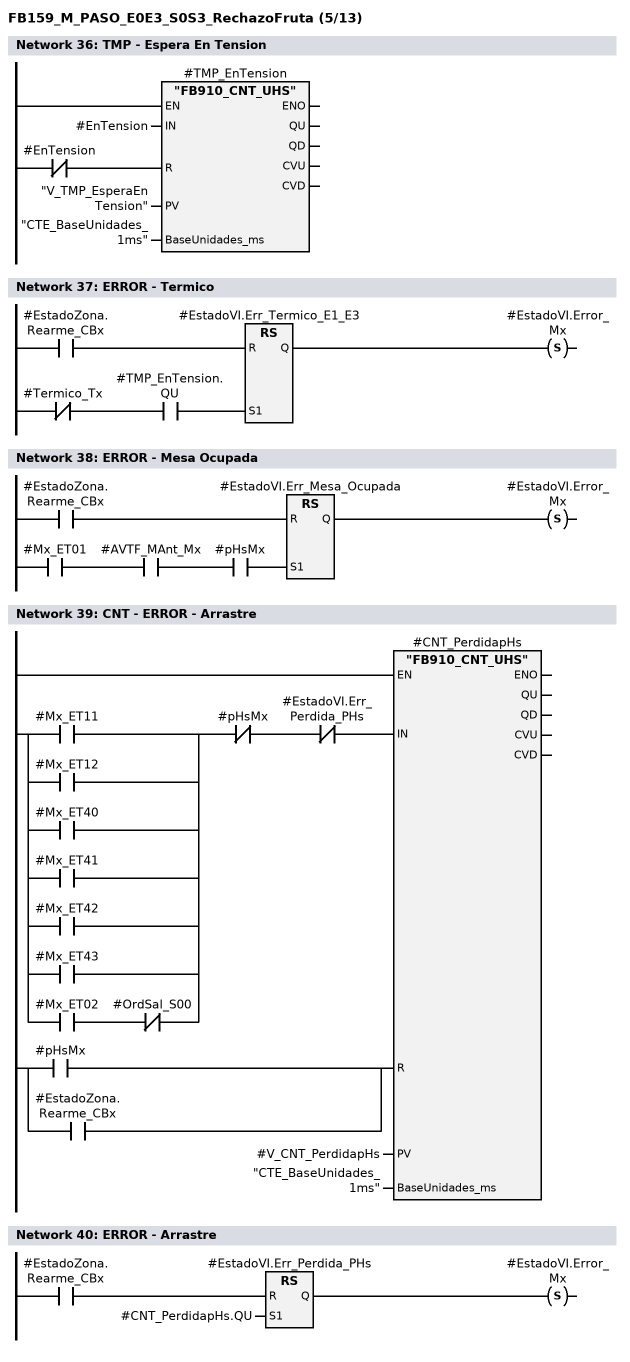
   RUNG wire#powerrail
      #TMP_EnTension(R := wire#w1, IN := #EnTension, PV := "V_TMP_EsperaEnTension", BaseUnidades_ms := "CTE_BaseUnidades_1ms", QU =>, QD =>, CVU =>, CVD =>)
   END_RUNG
   RUNG wire#powerrail
      I_Contact( #EnTension )
   END_RUNG wire#w1
   // the same network as SCL:
   #TMP_EnTension(IN := #EnTension,   // "FB910_CNT_UHS"
                  R := NOT #EnTension,
                  PV := "V_TMP_EsperaEnTension",
                  BaseUnidades_ms := "CTE_BaseUnidades_1ms");
END_REGION

REGION Network 37: ERROR - Termico
   RUNG wire#powerrail
      Contact( #EstadoZona.Rearme_CBx )
      S_RS(operand := #EstadoVI.Err_Termico_E1_E3, s1 := wire#w1)
      S_Coil( #EstadoVI.Error_Mx )
   END_RUNG
   RUNG wire#powerrail
      I_Contact( #Termico_Tx )
      Contact( #TMP_EnTension.QU )
   END_RUNG wire#w1
   // the same network as SCL:
   IF #EstadoZona.Rearme_CBx THEN
       #EstadoVI.Err_Termico_E1_E3 := FALSE;   // RS flip-flop
   END_IF;
   IF NOT #Termico_Tx AND #TMP_EnTension.QU THEN #EstadoVI.Err_Termico_E1_E3 := TRUE; END_IF;
   IF #EstadoVI.Err_Termico_E1_E3 THEN #EstadoVI.Error_Mx := TRUE; END_IF;
END_REGION

REGION Network 38: ERROR - Mesa Ocupada
   RUNG wire#powerrail
      Contact( #EstadoZona.Rearme_CBx )
      S_RS(operand := #EstadoVI.Err_Mesa_Ocupada, s1 := wire#w1)
      S_Coil( #EstadoVI.Error_Mx )
   END_RUNG
   RUNG wire#powerrail
      Contact( #Mx_ET01 )
      Contact( #AVTF_MAnt_Mx )
      Contact( #pHsMx )
   END_RUNG wire#w1
   // the same network as SCL:
   IF #EstadoZona.Rearme_CBx THEN
       #EstadoVI.Err_Mesa_Ocupada := FALSE;   // RS flip-flop
   END_IF;
   IF #Mx_ET01 AND #AVTF_MAnt_Mx AND #pHsMx THEN #EstadoVI.Err_Mesa_Ocupada := TRUE; END_IF;
   IF #EstadoVI.Err_Mesa_Ocupada THEN #EstadoVI.Error_Mx := TRUE; END_IF;
END_REGION

REGION Network 39: CNT - ERROR - Arrastre
   RUNG wire#powerrail
      #CNT_PerdidapHs(IN := wire#w2, R := wire#w3, PV := #V_CNT_PerdidapHs, BaseUnidades_ms := "CTE_BaseUnidades_1ms", QU =>, QD =>, CVU =>, CVD =>)
   END_RUNG
   RUNG wire#powerrail
      Contact( #Mx_ET11 )
      wire#w1
      I_Contact( #pHsMx )
      I_Contact( #EstadoVI.Err_Perdida_PHs )
   END_RUNG wire#w2
   RUNG wire#powerrail
      Contact( #Mx_ET12 )
   END_RUNG wire#w1
   RUNG wire#powerrail
      Contact( #Mx_ET40 )
   END_RUNG wire#w1
   RUNG wire#powerrail
      Contact( #Mx_ET41 )
   END_RUNG wire#w1
   RUNG wire#powerrail
      Contact( #Mx_ET42 )
   END_RUNG wire#w1
   RUNG wire#powerrail
      Contact( #Mx_ET43 )
   END_RUNG wire#w1
   RUNG wire#powerrail
      Contact( #Mx_ET02 )
      I_Contact( #OrdSal_S00 )
   END_RUNG wire#w1
   RUNG wire#powerrail
      Contact( #pHsMx )
   END_RUNG wire#w3
   RUNG wire#powerrail
      Contact( #EstadoZona.Rearme_CBx )
   END_RUNG wire#w3
   // the same network as SCL:
   #CNT_PerdidapHs(IN := (#Mx_ET11 OR #Mx_ET12 OR #Mx_ET40 OR #Mx_ET41 OR #Mx_ET42 OR #Mx_ET43 OR (#Mx_ET02 AND NOT #OrdSal_S00)) AND NOT #pHsMx AND NOT #EstadoVI.Err_Perdida_PHs,   // "FB910_CNT_UHS"
                   R := #pHsMx OR #EstadoZona.Rearme_CBx,
                   PV := #V_CNT_PerdidapHs,
                   BaseUnidades_ms := "CTE_BaseUnidades_1ms");
END_REGION

REGION Network 40: ERROR - Arrastre
   RUNG wire#powerrail
      Contact( #EstadoZona.Rearme_CBx )
      S_RS(operand := #EstadoVI.Err_Perdida_PHs, s1 := #CNT_PerdidapHs.QU)
      S_Coil( #EstadoVI.Error_Mx )
   END_RUNG
   // the same network as SCL:
   IF #EstadoZona.Rearme_CBx THEN
       #EstadoVI.Err_Perdida_PHs := FALSE;   // RS flip-flop
   END_IF;
   IF #CNT_PerdidapHs.QU THEN #EstadoVI.Err_Perdida_PHs := TRUE; END_IF;
   IF #EstadoVI.Err_Perdida_PHs THEN #EstadoVI.Error_Mx := TRUE; END_IF;
END_REGION

REGION Network 41: ERROR - Descarga por S3
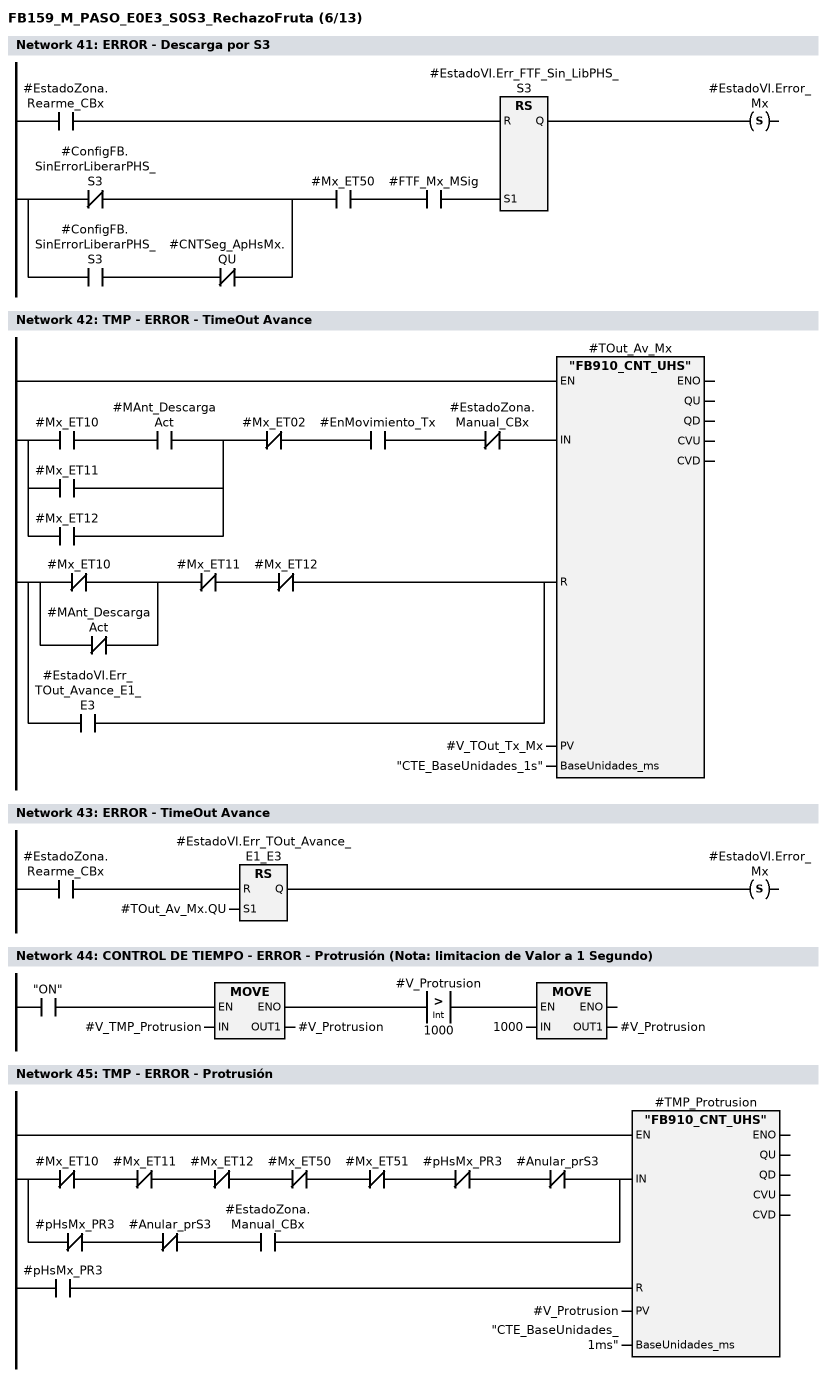
   RUNG wire#powerrail
      Contact( #EstadoZona.Rearme_CBx )
      S_RS(operand := #EstadoVI.Err_FTF_Sin_LibPHS_S3, s1 := wire#w2)
      S_Coil( #EstadoVI.Error_Mx )
   END_RUNG
   RUNG wire#powerrail
      I_Contact( #ConfigFB.SinErrorLiberarPHS_S3 )
      wire#w1
      Contact( #Mx_ET50 )
      Contact( #FTF_Mx_MSig )
   END_RUNG wire#w2
   RUNG wire#powerrail
      Contact( #ConfigFB.SinErrorLiberarPHS_S3 )
      I_Contact( #CNTSeg_ApHsMx.QU )
   END_RUNG wire#w1
   // the same network as SCL:
   IF #EstadoZona.Rearme_CBx THEN
       #EstadoVI.Err_FTF_Sin_LibPHS_S3 := FALSE;   // RS flip-flop
   END_IF;
   IF (NOT #ConfigFB.SinErrorLiberarPHS_S3 OR (#ConfigFB.SinErrorLiberarPHS_S3 AND NOT #CNTSeg_ApHsMx.QU)) AND #Mx_ET50 AND #FTF_Mx_MSig THEN
       #EstadoVI.Err_FTF_Sin_LibPHS_S3 := TRUE;
   END_IF;
   IF #EstadoVI.Err_FTF_Sin_LibPHS_S3 THEN #EstadoVI.Error_Mx := TRUE; END_IF;
END_REGION

REGION Network 42: TMP - ERROR - TimeOut Avance
   RUNG wire#powerrail
      #TOut_Av_Mx(IN := wire#w2, R := wire#w4, PV := #V_TOut_Tx_Mx, BaseUnidades_ms := "CTE_BaseUnidades_1s", QU =>, QD =>, CVU =>, CVD =>)
   END_RUNG
   RUNG wire#powerrail
      Contact( #Mx_ET10 )
      Contact( #MAnt_DescargaAct )
      wire#w1
      I_Contact( #Mx_ET02 )
      Contact( #EnMovimiento_Tx )
      I_Contact( #EstadoZona.Manual_CBx )
   END_RUNG wire#w2
   RUNG wire#powerrail
      Contact( #Mx_ET11 )
   END_RUNG wire#w1
   RUNG wire#powerrail
      Contact( #Mx_ET12 )
   END_RUNG wire#w1
   RUNG wire#powerrail
      I_Contact( #Mx_ET10 )
      wire#w3
      I_Contact( #Mx_ET11 )
      I_Contact( #Mx_ET12 )
   END_RUNG wire#w4
   RUNG wire#powerrail
      I_Contact( #MAnt_DescargaAct )
   END_RUNG wire#w3
   RUNG wire#powerrail
      Contact( #EstadoVI.Err_TOut_Avance_E1_E3 )
   END_RUNG wire#w4
   // the same network as SCL:
   #TOut_Av_Mx(IN := ((#Mx_ET10 AND #MAnt_DescargaAct) OR #Mx_ET11 OR #Mx_ET12) AND NOT #Mx_ET02 AND #EnMovimiento_Tx AND NOT #EstadoZona.Manual_CBx,   // "FB910_CNT_UHS"
               R := ((NOT #Mx_ET10 OR NOT #MAnt_DescargaAct) AND NOT #Mx_ET11 AND NOT #Mx_ET12) OR #EstadoVI.Err_TOut_Avance_E1_E3,
               PV := #V_TOut_Tx_Mx,
               BaseUnidades_ms := "CTE_BaseUnidades_1s");
END_REGION

REGION Network 43: ERROR - TimeOut Avance
   RUNG wire#powerrail
      Contact( #EstadoZona.Rearme_CBx )
      S_RS(operand := #EstadoVI.Err_TOut_Avance_E1_E3, s1 := #TOut_Av_Mx.QU)
      S_Coil( #EstadoVI.Error_Mx )
   END_RUNG
   // the same network as SCL:
   IF #EstadoZona.Rearme_CBx THEN
       #EstadoVI.Err_TOut_Avance_E1_E3 := FALSE;   // RS flip-flop
   END_IF;
   IF #TOut_Av_Mx.QU THEN #EstadoVI.Err_TOut_Avance_E1_E3 := TRUE; END_IF;
   IF #EstadoVI.Err_TOut_Avance_E1_E3 THEN #EstadoVI.Error_Mx := TRUE; END_IF;
END_REGION

REGION Network 44: CONTROL DE TIEMPO - ERROR - Protrusión (Nota: limitacion de Valor a 1 Segundo)
   RUNG wire#powerrail
      Contact( "ON" )
      Move(in := #V_TMP_Protrusion, out1 => #V_Protrusion)
      { S7_Templates := "SrcType := Int" } GT_Contact(in1 := #V_Protrusion, in2 := 1000)
      Move(in := 1000, out1 => #V_Protrusion)
   END_RUNG
   // the same network as SCL:
   IF "ON" THEN #V_Protrusion := #V_TMP_Protrusion; END_IF;
   IF "ON" AND (#V_Protrusion > 1000) THEN #V_Protrusion := 1000; END_IF;
END_REGION

REGION Network 45: TMP - ERROR - Protrusión
   RUNG wire#powerrail
      #TMP_Protrusion(IN := wire#w1, R := wire#w2, PV := #V_Protrusion, BaseUnidades_ms := "CTE_BaseUnidades_1ms", QU =>, QD =>, CVU =>, CVD =>)
   END_RUNG
   RUNG wire#powerrail
      I_Contact( #Mx_ET10 )
      I_Contact( #Mx_ET11 )
      I_Contact( #Mx_ET12 )
      I_Contact( #Mx_ET50 )
      I_Contact( #Mx_ET51 )
      I_Contact( #pHsMx_PR3 )
      I_Contact( #Anular_prS3 )
   END_RUNG wire#w1
   RUNG wire#powerrail
      I_Contact( #pHsMx_PR3 )
      I_Contact( #Anular_prS3 )
      Contact( #EstadoZona.Manual_CBx )
   END_RUNG wire#w1
   RUNG wire#powerrail
      Contact( #pHsMx_PR3 )
   END_RUNG wire#w2
   // the same network as SCL:
   #TMP_Protrusion(IN := (NOT #Mx_ET10 AND NOT #Mx_ET11 AND NOT #Mx_ET12 AND NOT #Mx_ET50 AND NOT #Mx_ET51 AND NOT #pHsMx_PR3 AND NOT #Anular_prS3) OR (NOT #pHsMx_PR3 AND NOT #Anular_prS3 AND #EstadoZona.Manual_CBx),   // "FB910_CNT_UHS"
                   R := #pHsMx_PR3,
                   PV := #V_Protrusion,
                   BaseUnidades_ms := "CTE_BaseUnidades_1ms");
END_REGION

REGION Network 46: ERROR - Protrusión
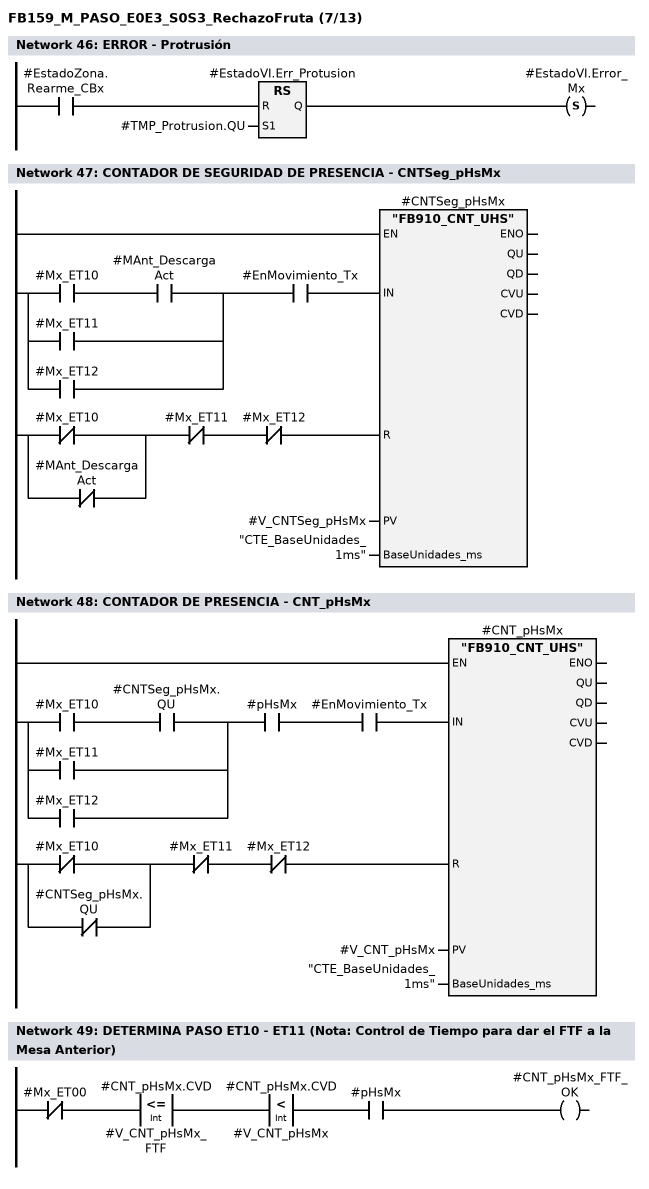
   RUNG wire#powerrail
      Contact( #EstadoZona.Rearme_CBx )
      S_RS(operand := #EstadoVI.Err_Protusion, s1 := #TMP_Protrusion.QU)
      S_Coil( #EstadoVI.Error_Mx )
   END_RUNG
   // the same network as SCL:
   IF #EstadoZona.Rearme_CBx THEN
       #EstadoVI.Err_Protusion := FALSE;   // RS flip-flop
   END_IF;
   IF #TMP_Protrusion.QU THEN #EstadoVI.Err_Protusion := TRUE; END_IF;
   IF #EstadoVI.Err_Protusion THEN #EstadoVI.Error_Mx := TRUE; END_IF;
END_REGION

REGION Network 47: CONTADOR DE SEGURIDAD DE PRESENCIA - CNTSeg_pHsMx
   RUNG wire#powerrail
      #CNTSeg_pHsMx(IN := wire#w2, R := wire#w4, PV := #V_CNTSeg_pHsMx, BaseUnidades_ms := "CTE_BaseUnidades_1ms", QU =>, QD =>, CVU =>, CVD =>)
   END_RUNG
   RUNG wire#powerrail
      Contact( #Mx_ET10 )
      Contact( #MAnt_DescargaAct )
      wire#w1
      Contact( #EnMovimiento_Tx )
   END_RUNG wire#w2
   RUNG wire#powerrail
      Contact( #Mx_ET11 )
   END_RUNG wire#w1
   RUNG wire#powerrail
      Contact( #Mx_ET12 )
   END_RUNG wire#w1
   RUNG wire#powerrail
      I_Contact( #Mx_ET10 )
      wire#w3
      I_Contact( #Mx_ET11 )
      I_Contact( #Mx_ET12 )
   END_RUNG wire#w4
   RUNG wire#powerrail
      I_Contact( #MAnt_DescargaAct )
   END_RUNG wire#w3
   // the same network as SCL:
   #CNTSeg_pHsMx(IN := ((#Mx_ET10 AND #MAnt_DescargaAct) OR #Mx_ET11 OR #Mx_ET12) AND #EnMovimiento_Tx,   // "FB910_CNT_UHS"
                 R := (NOT #Mx_ET10 OR NOT #MAnt_DescargaAct) AND NOT #Mx_ET11 AND NOT #Mx_ET12,
                 PV := #V_CNTSeg_pHsMx,
                 BaseUnidades_ms := "CTE_BaseUnidades_1ms");
END_REGION

REGION Network 48: CONTADOR DE PRESENCIA - CNT_pHsMx
   RUNG wire#powerrail
      #CNT_pHsMx(IN := wire#w2, R := wire#w4, PV := #V_CNT_pHsMx, BaseUnidades_ms := "CTE_BaseUnidades_1ms", QU =>, QD =>, CVU =>, CVD =>)
   END_RUNG
   RUNG wire#powerrail
      Contact( #Mx_ET10 )
      Contact( #CNTSeg_pHsMx.QU )
      wire#w1
      Contact( #pHsMx )
      Contact( #EnMovimiento_Tx )
   END_RUNG wire#w2
   RUNG wire#powerrail
      Contact( #Mx_ET11 )
   END_RUNG wire#w1
   RUNG wire#powerrail
      Contact( #Mx_ET12 )
   END_RUNG wire#w1
   RUNG wire#powerrail
      I_Contact( #Mx_ET10 )
      wire#w3
      I_Contact( #Mx_ET11 )
      I_Contact( #Mx_ET12 )
   END_RUNG wire#w4
   RUNG wire#powerrail
      I_Contact( #CNTSeg_pHsMx.QU )
   END_RUNG wire#w3
   // the same network as SCL:
   #CNT_pHsMx(IN := ((#Mx_ET10 AND #CNTSeg_pHsMx.QU) OR #Mx_ET11 OR #Mx_ET12) AND #pHsMx AND #EnMovimiento_Tx,   // "FB910_CNT_UHS"
              R := (NOT #Mx_ET10 OR NOT #CNTSeg_pHsMx.QU) AND NOT #Mx_ET11 AND NOT #Mx_ET12,
              PV := #V_CNT_pHsMx,
              BaseUnidades_ms := "CTE_BaseUnidades_1ms");
END_REGION

REGION Network 49: DETERMINA PASO ET10 - ET11 (Nota: Control de Tiempo para dar el FTF a la Mesa Anterior)
   RUNG wire#powerrail
      I_Contact( #Mx_ET00 )
      { S7_Templates := "SrcType := Int" } LE_Contact(in1 := #CNT_pHsMx.CVD, in2 := #V_CNT_pHsMx_FTF)
      { S7_Templates := "SrcType := Int" } LT_Contact(in1 := #CNT_pHsMx.CVD, in2 := #V_CNT_pHsMx)
      Contact( #pHsMx )
      Coil( #CNT_pHsMx_FTF_OK )
   END_RUNG
   // the same network as SCL:
   #CNT_pHsMx_FTF_OK := NOT #Mx_ET00 AND (#CNT_pHsMx.CVD <= #V_CNT_pHsMx_FTF) AND (#CNT_pHsMx.CVD < #V_CNT_pHsMx) AND #pHsMx;
END_REGION

REGION Network 50: CONTADOR SEGURIDAD DE AUSENCIA - CNTSeg_ApHsMx ??????? RESTAR VALOR DE POSICIONAMIENTO
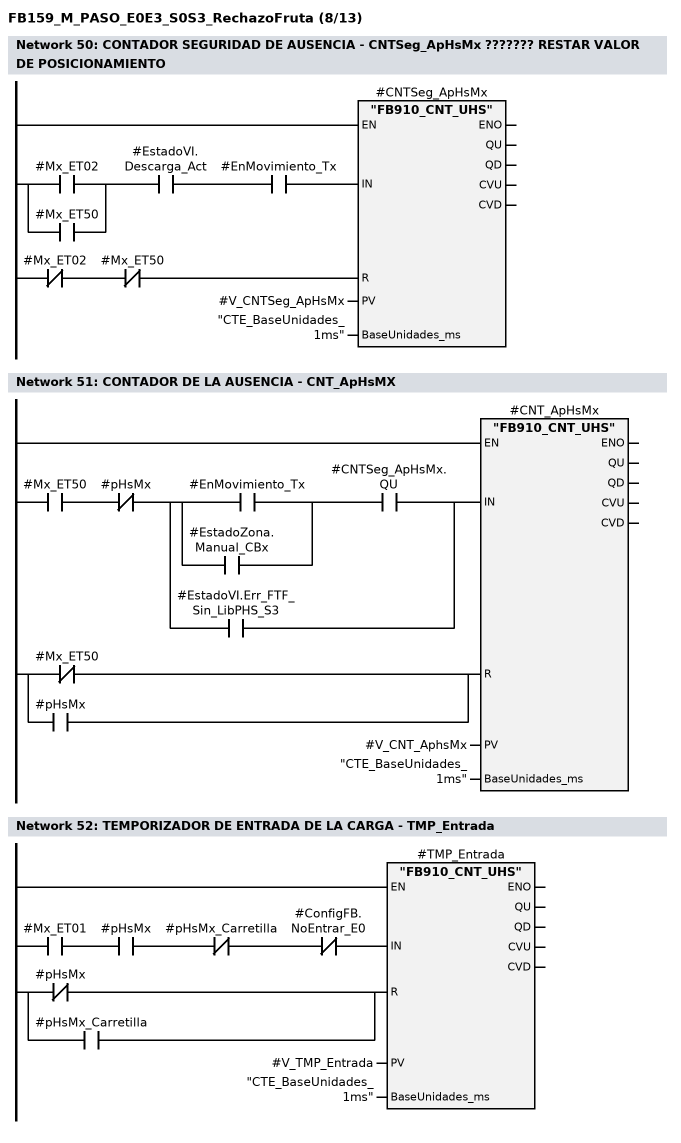
   RUNG wire#powerrail
      #CNTSeg_ApHsMx(IN := wire#w2, R := wire#w3, PV := #V_CNTSeg_ApHsMx, BaseUnidades_ms := "CTE_BaseUnidades_1ms", QU =>, QD =>, CVU =>, CVD =>)
   END_RUNG
   RUNG wire#powerrail
      Contact( #Mx_ET02 )
      wire#w1
      Contact( #EstadoVI.Descarga_Act )
      Contact( #EnMovimiento_Tx )
   END_RUNG wire#w2
   RUNG wire#powerrail
      Contact( #Mx_ET50 )
   END_RUNG wire#w1
   RUNG wire#powerrail
      I_Contact( #Mx_ET02 )
      I_Contact( #Mx_ET50 )
   END_RUNG wire#w3
   // the same network as SCL:
   #CNTSeg_ApHsMx(IN := (#Mx_ET02 OR #Mx_ET50) AND #EstadoVI.Descarga_Act AND #EnMovimiento_Tx,   // "FB910_CNT_UHS"
                  R := NOT #Mx_ET02 AND NOT #Mx_ET50,
                  PV := #V_CNTSeg_ApHsMx,
                  BaseUnidades_ms := "CTE_BaseUnidades_1ms");
END_REGION

REGION Network 51: CONTADOR DE LA AUSENCIA - CNT_ApHsMX
   RUNG wire#powerrail
      #CNT_ApHsMx(IN := wire#w3, R := wire#w4, PV := #V_CNT_AphsMx, BaseUnidades_ms := "CTE_BaseUnidades_1ms", QU =>, QD =>, CVU =>, CVD =>)
   END_RUNG
   RUNG wire#powerrail
      Contact( #Mx_ET50 )
      I_Contact( #pHsMx )
      wire#w1
      Contact( #EnMovimiento_Tx )
      wire#w2
      Contact( #CNTSeg_ApHsMx.QU )
   END_RUNG wire#w3
   RUNG wire#w1
      Contact( #EstadoZona.Manual_CBx )
   END_RUNG wire#w2
   RUNG wire#w1
      Contact( #EstadoVI.Err_FTF_Sin_LibPHS_S3 )
   END_RUNG wire#w3
   RUNG wire#powerrail
      I_Contact( #Mx_ET50 )
   END_RUNG wire#w4
   RUNG wire#powerrail
      Contact( #pHsMx )
   END_RUNG wire#w4
   // the same network as SCL:
   #CNT_ApHsMx(IN := #Mx_ET50 AND NOT #pHsMx AND (((#EnMovimiento_Tx OR #EstadoZona.Manual_CBx) AND #CNTSeg_ApHsMx.QU) OR #EstadoVI.Err_FTF_Sin_LibPHS_S3),   // "FB910_CNT_UHS"
               R := NOT #Mx_ET50 OR #pHsMx,
               PV := #V_CNT_AphsMx,
               BaseUnidades_ms := "CTE_BaseUnidades_1ms");
END_REGION

REGION Network 52: TEMPORIZADOR DE ENTRADA DE LA CARGA - TMP_Entrada
   RUNG wire#powerrail
      #TMP_Entrada(IN := wire#w1, R := wire#w2, PV := #V_TMP_Entrada, BaseUnidades_ms := "CTE_BaseUnidades_1ms", QU =>, QD =>, CVU =>, CVD =>)
   END_RUNG
   RUNG wire#powerrail
      Contact( #Mx_ET01 )
      Contact( #pHsMx )
      I_Contact( #pHsMx_Carretilla )
      I_Contact( #ConfigFB.NoEntrar_E0 )
   END_RUNG wire#w1
   RUNG wire#powerrail
      I_Contact( #pHsMx )
   END_RUNG wire#w2
   RUNG wire#powerrail
      Contact( #pHsMx_Carretilla )
   END_RUNG wire#w2
   // the same network as SCL:
   #TMP_Entrada(IN := #Mx_ET01 AND #pHsMx AND NOT #pHsMx_Carretilla AND NOT #ConfigFB.NoEntrar_E0,   // "FB910_CNT_UHS"
                R := NOT #pHsMx OR #pHsMx_Carretilla,
                PV := #V_TMP_Entrada,
                BaseUnidades_ms := "CTE_BaseUnidades_1ms");
END_REGION

REGION Network 53: CONTADOR PARA CENTRAJE - CNT_Centrado >> REPOSO
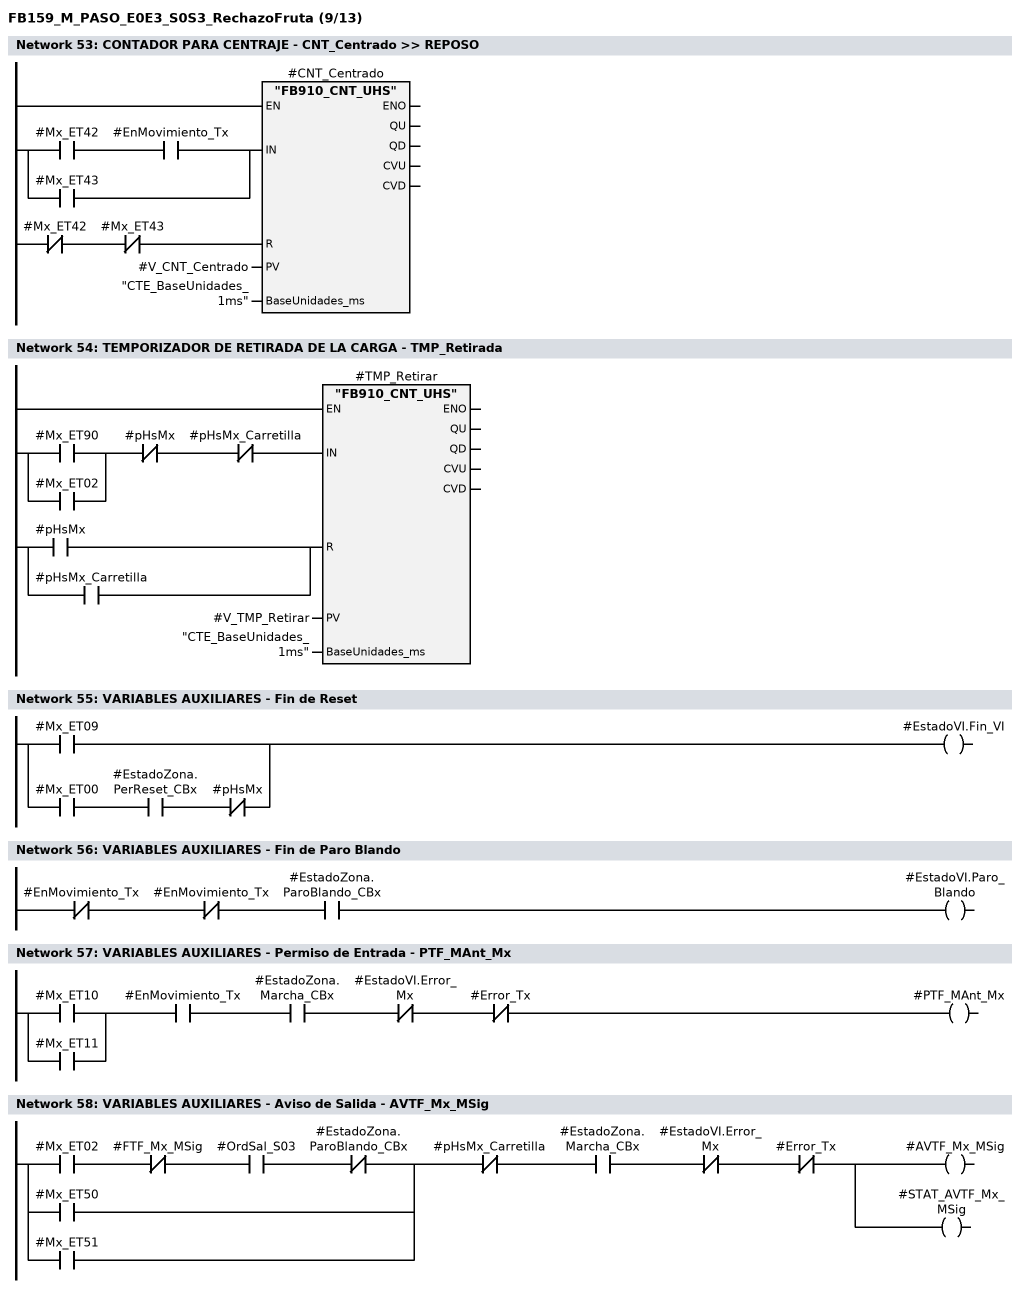
   RUNG wire#powerrail
      #CNT_Centrado(IN := wire#w1, R := wire#w2, PV := #V_CNT_Centrado, BaseUnidades_ms := "CTE_BaseUnidades_1ms", QU =>, QD =>, CVU =>, CVD =>)
   END_RUNG
   RUNG wire#powerrail
      Contact( #Mx_ET42 )
      Contact( #EnMovimiento_Tx )
   END_RUNG wire#w1
   RUNG wire#powerrail
      Contact( #Mx_ET43 )
   END_RUNG wire#w1
   RUNG wire#powerrail
      I_Contact( #Mx_ET42 )
      I_Contact( #Mx_ET43 )
   END_RUNG wire#w2
   // the same network as SCL:
   #CNT_Centrado(IN := (#Mx_ET42 AND #EnMovimiento_Tx) OR #Mx_ET43,   // "FB910_CNT_UHS"
                 R := NOT #Mx_ET42 AND NOT #Mx_ET43,
                 PV := #V_CNT_Centrado,
                 BaseUnidades_ms := "CTE_BaseUnidades_1ms");
END_REGION

REGION Network 54: TEMPORIZADOR DE RETIRADA DE LA CARGA - TMP_Retirada
   RUNG wire#powerrail
      #TMP_Retirar(IN := wire#w2, R := wire#w3, PV := #V_TMP_Retirar, BaseUnidades_ms := "CTE_BaseUnidades_1ms", QU =>, QD =>, CVU =>, CVD =>)
   END_RUNG
   RUNG wire#powerrail
      Contact( #Mx_ET90 )
      wire#w1
      I_Contact( #pHsMx )
      I_Contact( #pHsMx_Carretilla )
   END_RUNG wire#w2
   RUNG wire#powerrail
      Contact( #Mx_ET02 )
   END_RUNG wire#w1
   RUNG wire#powerrail
      Contact( #pHsMx )
   END_RUNG wire#w3
   RUNG wire#powerrail
      Contact( #pHsMx_Carretilla )
   END_RUNG wire#w3
   // the same network as SCL:
   #TMP_Retirar(IN := (#Mx_ET90 OR #Mx_ET02) AND NOT #pHsMx AND NOT #pHsMx_Carretilla,   // "FB910_CNT_UHS"
                R := #pHsMx OR #pHsMx_Carretilla,
                PV := #V_TMP_Retirar,
                BaseUnidades_ms := "CTE_BaseUnidades_1ms");
END_REGION

REGION Network 55: VARIABLES AUXILIARES - Fin de Reset
   RUNG wire#powerrail
      Contact( #Mx_ET09 )
      wire#w1
      Coil( #EstadoVI.Fin_VI )
   END_RUNG
   RUNG wire#powerrail
      Contact( #Mx_ET00 )
      Contact( #EstadoZona.PerReset_CBx )
      I_Contact( #pHsMx )
   END_RUNG wire#w1
   // the same network as SCL:
   #EstadoVI.Fin_VI := #Mx_ET09 OR (#Mx_ET00 AND #EstadoZona.PerReset_CBx AND NOT #pHsMx);
END_REGION

REGION Network 56: VARIABLES AUXILIARES - Fin de Paro Blando
   RUNG wire#powerrail
      I_Contact( #EnMovimiento_Tx )
      I_Contact( #EnMovimiento_Tx )
      Contact( #EstadoZona.ParoBlando_CBx )
      Coil( #EstadoVI.Paro_Blando )
   END_RUNG
   // the same network as SCL:
   #EstadoVI.Paro_Blando := NOT #EnMovimiento_Tx AND NOT #EnMovimiento_Tx AND #EstadoZona.ParoBlando_CBx;
END_REGION

REGION Network 57: VARIABLES AUXILIARES - Permiso de Entrada - PTF_MAnt_Mx
   RUNG wire#powerrail
      Contact( #Mx_ET10 )
      wire#w1
      Contact( #EnMovimiento_Tx )
      Contact( #EstadoZona.Marcha_CBx )
      I_Contact( #EstadoVI.Error_Mx )
      I_Contact( #Error_Tx )
      Coil( #PTF_MAnt_Mx )
   END_RUNG
   RUNG wire#powerrail
      Contact( #Mx_ET11 )
   END_RUNG wire#w1
   // the same network as SCL:
   #PTF_MAnt_Mx := (#Mx_ET10 OR #Mx_ET11) AND #EnMovimiento_Tx AND #EstadoZona.Marcha_CBx AND NOT #EstadoVI.Error_Mx AND NOT #Error_Tx;
END_REGION

REGION Network 58: VARIABLES AUXILIARES - Aviso de Salida - AVTF_Mx_MSig
   RUNG wire#powerrail
      Contact( #Mx_ET02 )
      I_Contact( #FTF_Mx_MSig )
      Contact( #OrdSal_S03 )
      I_Contact( #EstadoZona.ParoBlando_CBx )
      wire#w1
      I_Contact( #pHsMx_Carretilla )
      Contact( #EstadoZona.Marcha_CBx )
      I_Contact( #EstadoVI.Error_Mx )
      I_Contact( #Error_Tx )
      wire#w2
      Coil( #AVTF_Mx_MSig )
   END_RUNG
   RUNG wire#powerrail
      Contact( #Mx_ET50 )
   END_RUNG wire#w1
   RUNG wire#powerrail
      Contact( #Mx_ET51 )
   END_RUNG wire#w1
   RUNG wire#w2
      Coil( #STAT_AVTF_Mx_MSig )
   END_RUNG
   // the same network as SCL:
   #AVTF_Mx_MSig := ((#Mx_ET02 AND NOT #FTF_Mx_MSig AND #OrdSal_S03 AND NOT #EstadoZona.ParoBlando_CBx) OR #Mx_ET50 OR #Mx_ET51) AND NOT #pHsMx_Carretilla AND #EstadoZona.Marcha_CBx AND NOT #EstadoVI.Error_Mx AND NOT #Error_Tx;
   #STAT_AVTF_Mx_MSig := #AVTF_Mx_MSig;
END_REGION

REGION Network 59: VARIABLES AUXILIARES - P_Mens_Mx_MSig (Nota: solo en ET51)
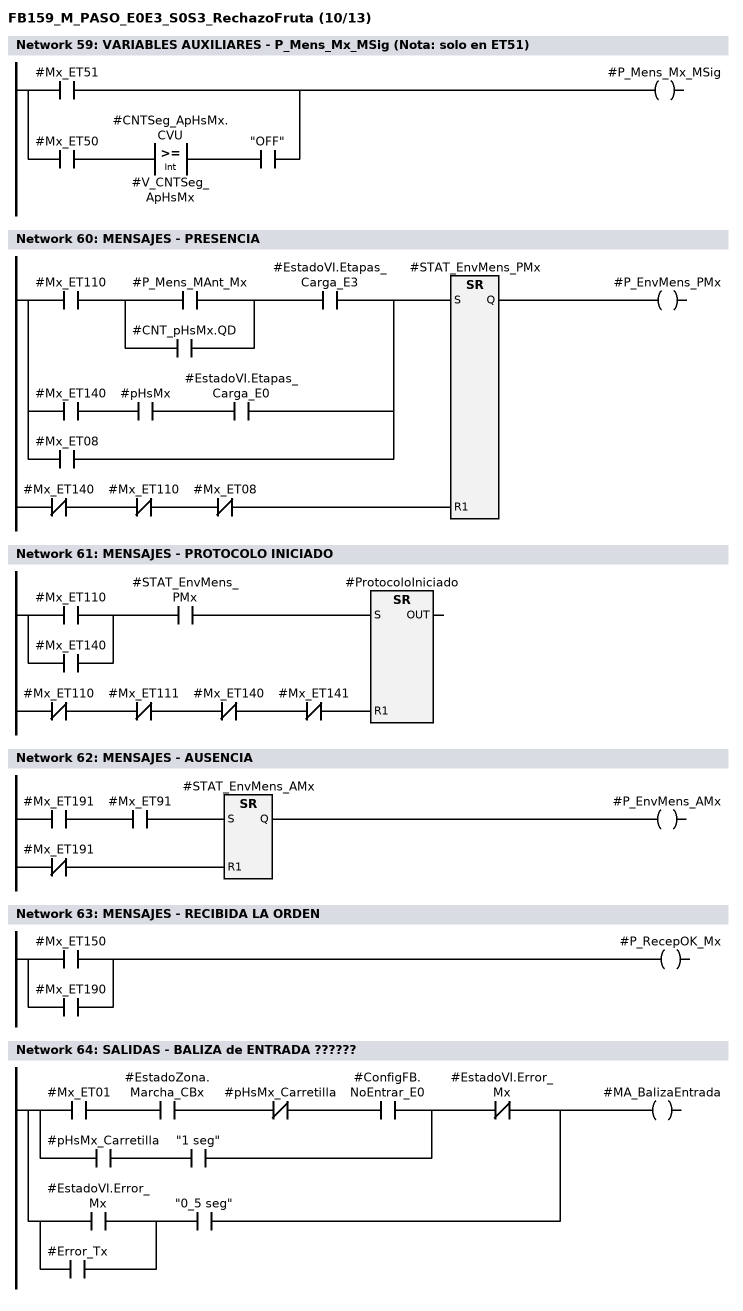
   RUNG wire#powerrail
      Contact( #Mx_ET51 )
      wire#w1
      Coil( #P_Mens_Mx_MSig )
   END_RUNG
   RUNG wire#powerrail
      Contact( #Mx_ET50 )
      { S7_Templates := "SrcType := Int" } GE_Contact(in1 := #CNTSeg_ApHsMx.CVU, in2 := #V_CNTSeg_ApHsMx)
      Contact( "OFF" )
   END_RUNG wire#w1
   // the same network as SCL:
   #P_Mens_Mx_MSig := #Mx_ET51 OR (#Mx_ET50 AND (#CNTSeg_ApHsMx.CVU >= #V_CNTSeg_ApHsMx) AND "OFF");
END_REGION

REGION Network 60: MENSAJES - PRESENCIA
   RUNG wire#powerrail
      Contact( #Mx_ET110 )
      wire#w1
      Contact( #P_Mens_MAnt_Mx )
      wire#w2
      Contact( #EstadoVI.Etapas_Carga_E3 )
      wire#w3
      S_SR(operand := #STAT_EnvMens_PMx, r1 := wire#w4)
      Coil( #P_EnvMens_PMx )
   END_RUNG
   RUNG wire#w1
      Contact( #CNT_pHsMx.QD )
   END_RUNG wire#w2
   RUNG wire#powerrail
      Contact( #Mx_ET140 )
      Contact( #pHsMx )
      Contact( #EstadoVI.Etapas_Carga_E0 )
   END_RUNG wire#w3
   RUNG wire#powerrail
      Contact( #Mx_ET08 )
   END_RUNG wire#w3
   RUNG wire#powerrail
      I_Contact( #Mx_ET140 )
      I_Contact( #Mx_ET110 )
      I_Contact( #Mx_ET08 )
   END_RUNG wire#w4
   // the same network as SCL:
   IF (#Mx_ET110 AND (#P_Mens_MAnt_Mx OR #CNT_pHsMx.QD) AND #EstadoVI.Etapas_Carga_E3) OR (#Mx_ET140 AND #pHsMx AND #EstadoVI.Etapas_Carga_E0) OR #Mx_ET08 THEN
       #STAT_EnvMens_PMx := TRUE;   // SR flip-flop
   END_IF;
   IF NOT #Mx_ET140 AND NOT #Mx_ET110 AND NOT #Mx_ET08 THEN #STAT_EnvMens_PMx := FALSE; END_IF;
   #P_EnvMens_PMx := #STAT_EnvMens_PMx;
END_REGION

REGION Network 61: MENSAJES - PROTOCOLO INICIADO
   RUNG wire#powerrail
      Contact( #Mx_ET110 )
      wire#w1
      Contact( #STAT_EnvMens_PMx )
      S_SR(operand := #ProtocoloIniciado, r1 := wire#w2)
   END_RUNG
   RUNG wire#powerrail
      Contact( #Mx_ET140 )
   END_RUNG wire#w1
   RUNG wire#powerrail
      I_Contact( #Mx_ET110 )
      I_Contact( #Mx_ET111 )
      I_Contact( #Mx_ET140 )
      I_Contact( #Mx_ET141 )
   END_RUNG wire#w2
   // the same network as SCL:
   IF (#Mx_ET110 OR #Mx_ET140) AND #STAT_EnvMens_PMx THEN
       #ProtocoloIniciado := TRUE;   // SR flip-flop
   END_IF;
   IF NOT #Mx_ET110 AND NOT #Mx_ET111 AND NOT #Mx_ET140 AND NOT #Mx_ET141 THEN
       #ProtocoloIniciado := FALSE;
   END_IF;
END_REGION

REGION Network 62: MENSAJES - AUSENCIA
   RUNG wire#powerrail
      Contact( #Mx_ET191 )
      Contact( #Mx_ET91 )
      S_SR(operand := #STAT_EnvMens_AMx, r1 := wire#w1)
      Coil( #P_EnvMens_AMx )
   END_RUNG
   RUNG wire#powerrail
      I_Contact( #Mx_ET191 )
   END_RUNG wire#w1
   // the same network as SCL:
   IF #Mx_ET191 AND #Mx_ET91 THEN
       #STAT_EnvMens_AMx := TRUE;   // SR flip-flop
   END_IF;
   IF NOT #Mx_ET191 THEN #STAT_EnvMens_AMx := FALSE; END_IF;
   #P_EnvMens_AMx := #STAT_EnvMens_AMx;
END_REGION

REGION Network 63: MENSAJES - RECIBIDA LA ORDEN
   RUNG wire#powerrail
      Contact( #Mx_ET150 )
      wire#w1
      Coil( #P_RecepOK_Mx )
   END_RUNG
   RUNG wire#powerrail
      Contact( #Mx_ET190 )
   END_RUNG wire#w1
   // the same network as SCL:
   #P_RecepOK_Mx := #Mx_ET150 OR #Mx_ET190;
END_REGION

REGION Network 64: SALIDAS - BALIZA de ENTRADA ??????
   RUNG wire#powerrail
      Contact( #Mx_ET01 )
      Contact( #EstadoZona.Marcha_CBx )
      I_Contact( #pHsMx_Carretilla )
      Contact( #ConfigFB.NoEntrar_E0 )
      wire#w1
      I_Contact( #EstadoVI.Error_Mx )
      wire#w2
      Coil( #MA_BalizaEntrada )
   END_RUNG
   RUNG wire#powerrail
      Contact( #pHsMx_Carretilla )
      Contact( "1 seg" )
   END_RUNG wire#w1
   RUNG wire#powerrail
      Contact( #EstadoVI.Error_Mx )
      wire#w3
      Contact( "0_5 seg" )
   END_RUNG wire#w2
   RUNG wire#powerrail
      Contact( #Error_Tx )
   END_RUNG wire#w3
   // the same network as SCL:
   #MA_BalizaEntrada := (((#Mx_ET01 AND #EstadoZona.Marcha_CBx AND NOT #pHsMx_Carretilla AND #ConfigFB.NoEntrar_E0) OR (#pHsMx_Carretilla AND "1 seg")) AND NOT #EstadoVI.Error_Mx) OR ((#EstadoVI.Error_Mx OR #Error_Tx) AND "0_5 seg");
END_REGION

REGION Network 65: SALIDAS - Avanzar E1E3
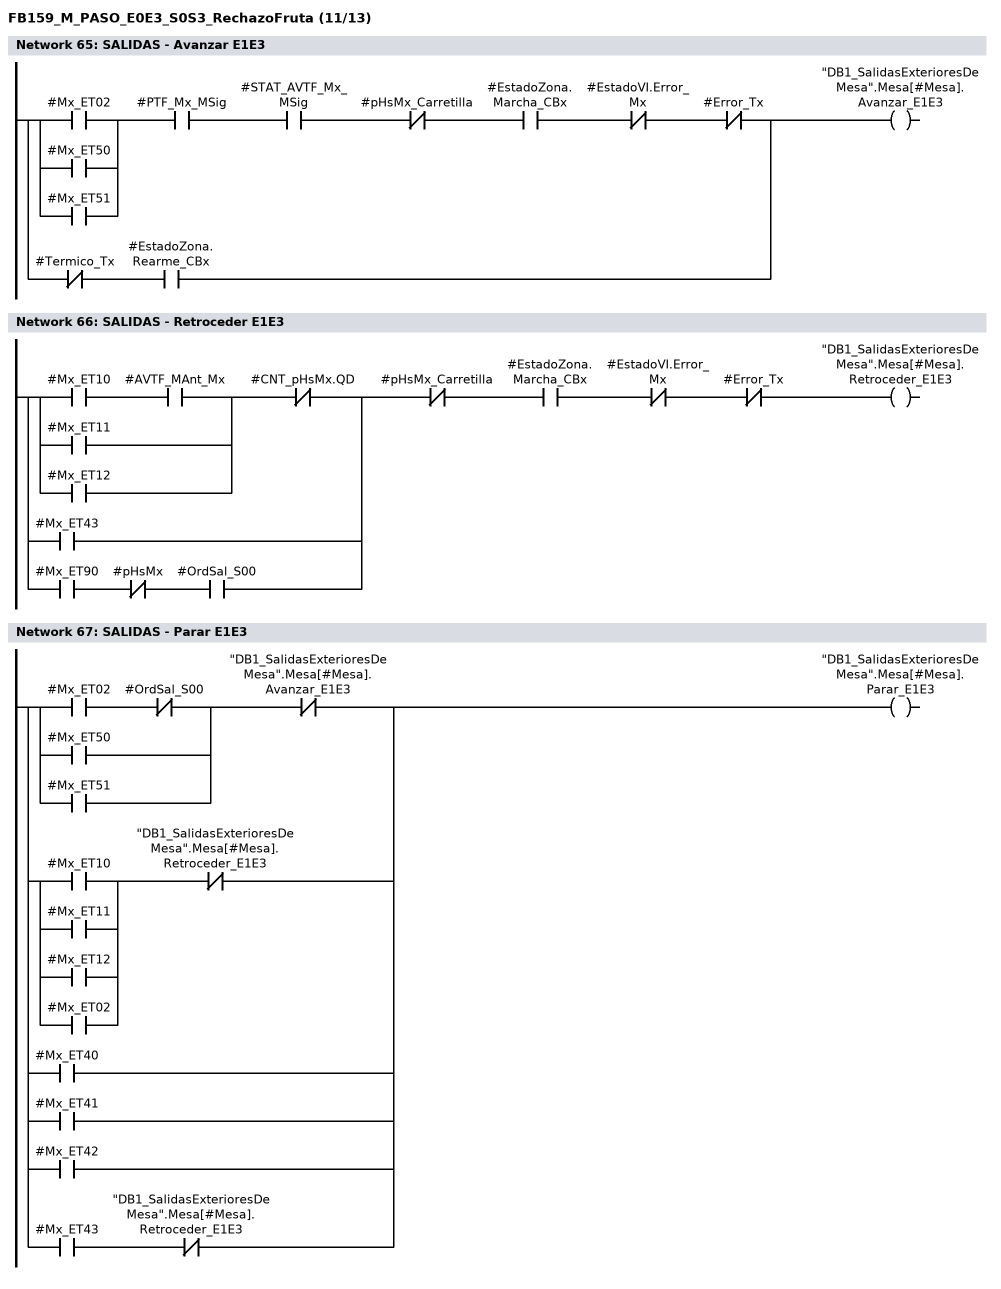
   RUNG wire#powerrail
      Contact( #Mx_ET02 )
      wire#w1
      Contact( #PTF_Mx_MSig )
      Contact( #STAT_AVTF_Mx_MSig )
      I_Contact( #pHsMx_Carretilla )
      Contact( #EstadoZona.Marcha_CBx )
      I_Contact( #EstadoVI.Error_Mx )
      I_Contact( #Error_Tx )
      wire#w2
      Coil( "DB1_SalidasExterioresDeMesa".Mesa[#Mesa].Avanzar_E1E3 )
   END_RUNG
   RUNG wire#powerrail
      Contact( #Mx_ET50 )
   END_RUNG wire#w1
   RUNG wire#powerrail
      Contact( #Mx_ET51 )
   END_RUNG wire#w1
   RUNG wire#powerrail
      I_Contact( #Termico_Tx )
      Contact( #EstadoZona.Rearme_CBx )
   END_RUNG wire#w2
   // the same network as SCL:
   "DB1_SalidasExterioresDeMesa".Mesa[#Mesa].Avanzar_E1E3 := ((#Mx_ET02 OR #Mx_ET50 OR #Mx_ET51) AND #PTF_Mx_MSig AND #STAT_AVTF_Mx_MSig AND NOT #pHsMx_Carretilla AND #EstadoZona.Marcha_CBx AND NOT #EstadoVI.Error_Mx AND NOT #Error_Tx) OR (NOT #Termico_Tx AND #EstadoZona.Rearme_CBx);
END_REGION

REGION Network 66: SALIDAS - Retroceder E1E3
   RUNG wire#powerrail
      Contact( #Mx_ET10 )
      Contact( #AVTF_MAnt_Mx )
      wire#w1
      I_Contact( #CNT_pHsMx.QD )
      wire#w2
      I_Contact( #pHsMx_Carretilla )
      Contact( #EstadoZona.Marcha_CBx )
      I_Contact( #EstadoVI.Error_Mx )
      I_Contact( #Error_Tx )
      Coil( "DB1_SalidasExterioresDeMesa".Mesa[#Mesa].Retroceder_E1E3 )
   END_RUNG
   RUNG wire#powerrail
      Contact( #Mx_ET11 )
   END_RUNG wire#w1
   RUNG wire#powerrail
      Contact( #Mx_ET12 )
   END_RUNG wire#w1
   RUNG wire#powerrail
      Contact( #Mx_ET43 )
   END_RUNG wire#w2
   RUNG wire#powerrail
      Contact( #Mx_ET90 )
      I_Contact( #pHsMx )
      Contact( #OrdSal_S00 )
   END_RUNG wire#w2
   // the same network as SCL:
   "DB1_SalidasExterioresDeMesa".Mesa[#Mesa].Retroceder_E1E3 := ((((#Mx_ET10 AND #AVTF_MAnt_Mx) OR #Mx_ET11 OR #Mx_ET12) AND NOT #CNT_pHsMx.QD) OR #Mx_ET43 OR (#Mx_ET90 AND NOT #pHsMx AND #OrdSal_S00)) AND NOT #pHsMx_Carretilla AND #EstadoZona.Marcha_CBx AND NOT #EstadoVI.Error_Mx AND NOT #Error_Tx;
END_REGION

REGION Network 67: SALIDAS - Parar E1E3
   RUNG wire#powerrail
      Contact( #Mx_ET02 )
      I_Contact( #OrdSal_S00 )
      wire#w1
      I_Contact( "DB1_SalidasExterioresDeMesa".Mesa[#Mesa].Avanzar_E1E3 )
      wire#w2
      Coil( "DB1_SalidasExterioresDeMesa".Mesa[#Mesa].Parar_E1E3 )
   END_RUNG
   RUNG wire#powerrail
      Contact( #Mx_ET50 )
   END_RUNG wire#w1
   RUNG wire#powerrail
      Contact( #Mx_ET51 )
   END_RUNG wire#w1
   RUNG wire#powerrail
      Contact( #Mx_ET10 )
      wire#w3
      I_Contact( "DB1_SalidasExterioresDeMesa".Mesa[#Mesa].Retroceder_E1E3 )
   END_RUNG wire#w2
   RUNG wire#powerrail
      Contact( #Mx_ET11 )
   END_RUNG wire#w3
   RUNG wire#powerrail
      Contact( #Mx_ET12 )
   END_RUNG wire#w3
   RUNG wire#powerrail
      Contact( #Mx_ET02 )
   END_RUNG wire#w3
   RUNG wire#powerrail
      Contact( #Mx_ET40 )
   END_RUNG wire#w2
   RUNG wire#powerrail
      Contact( #Mx_ET41 )
   END_RUNG wire#w2
   RUNG wire#powerrail
      Contact( #Mx_ET42 )
   END_RUNG wire#w2
   RUNG wire#powerrail
      Contact( #Mx_ET43 )
      I_Contact( "DB1_SalidasExterioresDeMesa".Mesa[#Mesa].Retroceder_E1E3 )
   END_RUNG wire#w2
   // the same network as SCL:
   "DB1_SalidasExterioresDeMesa".Mesa[#Mesa].Parar_E1E3 := (((#Mx_ET02 AND NOT #OrdSal_S00) OR #Mx_ET50 OR #Mx_ET51) AND NOT "DB1_SalidasExterioresDeMesa".Mesa[#Mesa].Avanzar_E1E3) OR ((#Mx_ET10 OR #Mx_ET11 OR #Mx_ET12 OR #Mx_ET02) AND NOT "DB1_SalidasExterioresDeMesa".Mesa[#Mesa].Retroceder_E1E3) OR #Mx_ET40 OR #Mx_ET41 OR #Mx_ET42 OR (#Mx_ET43 AND NOT "DB1_SalidasExterioresDeMesa".Mesa[#Mesa].Retroceder_E1E3);
END_REGION

REGION Network 68: SALIDAS - Valor Frecuencia Lenta E1E3
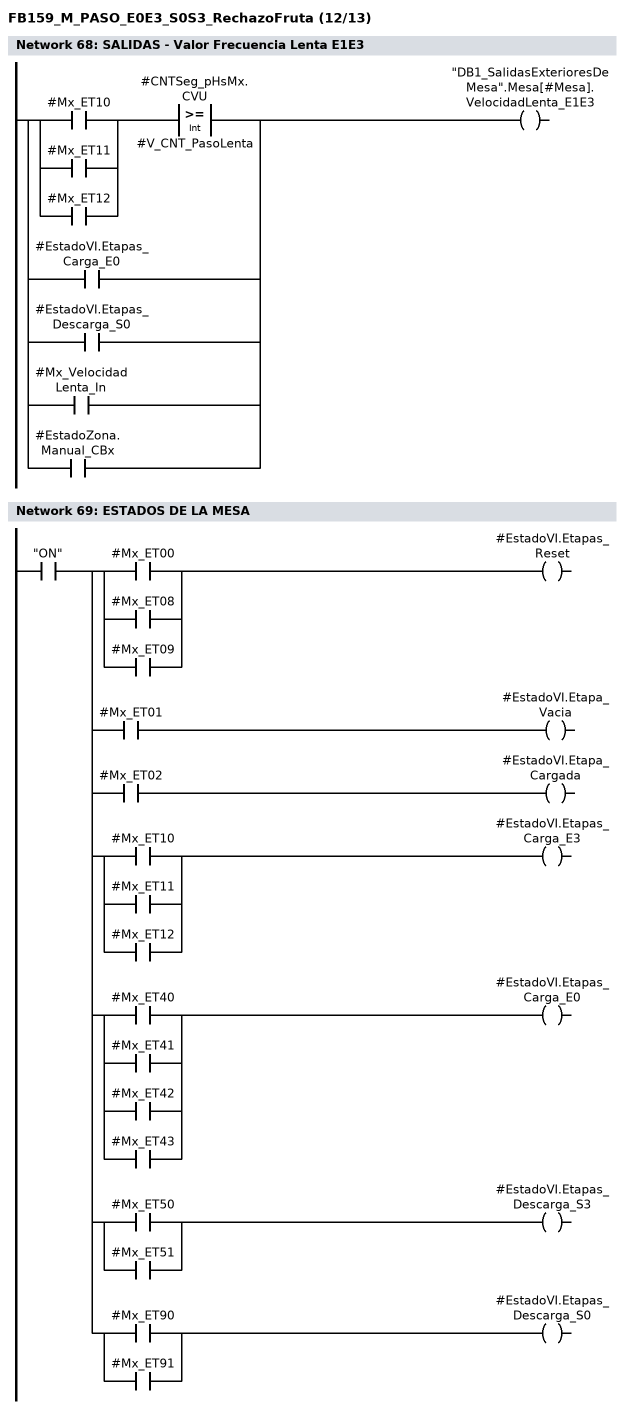
   RUNG wire#powerrail
      Contact( #Mx_ET10 )
      wire#w1
      { S7_Templates := "SrcType := Int" } GE_Contact(in1 := #CNTSeg_pHsMx.CVU, in2 := #V_CNT_PasoLenta)
      wire#w2
      Coil( "DB1_SalidasExterioresDeMesa".Mesa[#Mesa].VelocidadLenta_E1E3 )
   END_RUNG
   RUNG wire#powerrail
      Contact( #Mx_ET11 )
   END_RUNG wire#w1
   RUNG wire#powerrail
      Contact( #Mx_ET12 )
   END_RUNG wire#w1
   RUNG wire#powerrail
      Contact( #EstadoVI.Etapas_Carga_E0 )
   END_RUNG wire#w2
   RUNG wire#powerrail
      Contact( #EstadoVI.Etapas_Descarga_S0 )
   END_RUNG wire#w2
   RUNG wire#powerrail
      Contact( #Mx_VelocidadLenta_In )
   END_RUNG wire#w2
   RUNG wire#powerrail
      Contact( #EstadoZona.Manual_CBx )
   END_RUNG wire#w2
   // the same network as SCL:
   "DB1_SalidasExterioresDeMesa".Mesa[#Mesa].VelocidadLenta_E1E3 := ((#Mx_ET10 OR #Mx_ET11 OR #Mx_ET12) AND (#CNTSeg_pHsMx.CVU >= #V_CNT_PasoLenta)) OR #EstadoVI.Etapas_Carga_E0 OR #EstadoVI.Etapas_Descarga_S0 OR #Mx_VelocidadLenta_In OR #EstadoZona.Manual_CBx;
END_REGION

REGION Network 69: ESTADOS DE LA MESA
   RUNG wire#powerrail
      Contact( "ON" )
      wire#w1
      Contact( #Mx_ET00 )
      wire#w2
      Coil( #EstadoVI.Etapas_Reset )
   END_RUNG
   RUNG wire#w1
      Contact( #Mx_ET08 )
   END_RUNG wire#w2
   RUNG wire#w1
      Contact( #Mx_ET09 )
   END_RUNG wire#w2
   RUNG wire#w1
      Contact( #Mx_ET01 )
      Coil( #EstadoVI.Etapa_Vacia )
   END_RUNG
   RUNG wire#w1
      Contact( #Mx_ET02 )
      Coil( #EstadoVI.Etapa_Cargada )
   END_RUNG
   RUNG wire#w1
      Contact( #Mx_ET10 )
      wire#w3
      Coil( #EstadoVI.Etapas_Carga_E3 )
   END_RUNG
   RUNG wire#w1
      Contact( #Mx_ET11 )
   END_RUNG wire#w3
   RUNG wire#w1
      Contact( #Mx_ET12 )
   END_RUNG wire#w3
   RUNG wire#w1
      Contact( #Mx_ET40 )
      wire#w4
      Coil( #EstadoVI.Etapas_Carga_E0 )
   END_RUNG
   RUNG wire#w1
      Contact( #Mx_ET41 )
   END_RUNG wire#w4
   RUNG wire#w1
      Contact( #Mx_ET42 )
   END_RUNG wire#w4
   RUNG wire#w1
      Contact( #Mx_ET43 )
   END_RUNG wire#w4
   RUNG wire#w1
      Contact( #Mx_ET50 )
      wire#w5
      Coil( #EstadoVI.Etapas_Descarga_S3 )
   END_RUNG
   RUNG wire#w1
      Contact( #Mx_ET51 )
   END_RUNG wire#w5
   RUNG wire#w1
      Contact( #Mx_ET90 )
      wire#w6
      Coil( #EstadoVI.Etapas_Descarga_S0 )
   END_RUNG
   RUNG wire#w1
      Contact( #Mx_ET91 )
   END_RUNG wire#w6
   // the same network as SCL:
   #EstadoVI.Etapas_Reset := "ON" AND (#Mx_ET00 OR #Mx_ET08 OR #Mx_ET09);
   #EstadoVI.Etapa_Vacia := "ON" AND #Mx_ET01;
   #EstadoVI.Etapa_Cargada := "ON" AND #Mx_ET02;
   #EstadoVI.Etapas_Carga_E3 := "ON" AND (#Mx_ET10 OR #Mx_ET11 OR #Mx_ET12);
   #EstadoVI.Etapas_Carga_E0 := "ON" AND (#Mx_ET40 OR #Mx_ET41 OR #Mx_ET42 OR #Mx_ET43);
   #EstadoVI.Etapas_Descarga_S3 := "ON" AND (#Mx_ET50 OR #Mx_ET51);
   #EstadoVI.Etapas_Descarga_S0 := "ON" AND (#Mx_ET90 OR #Mx_ET91);
END_REGION

REGION Network 70: ENTRADAS DE LA MESA
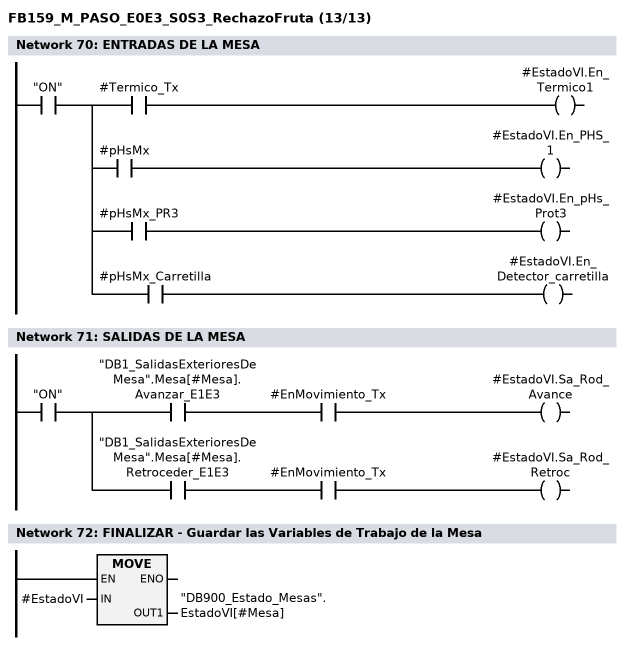
   RUNG wire#powerrail
      Contact( "ON" )
      wire#w1
      Contact( #Termico_Tx )
      Coil( #EstadoVI.En_Termico1 )
   END_RUNG
   RUNG wire#w1
      Contact( #pHsMx )
      Coil( #EstadoVI.En_PHS_1 )
   END_RUNG
   RUNG wire#w1
      Contact( #pHsMx_PR3 )
      Coil( #EstadoVI.En_pHs_Prot3 )
   END_RUNG
   RUNG wire#w1
      Contact( #pHsMx_Carretilla )
      Coil( #EstadoVI.En_Detector_carretilla )
   END_RUNG
   // the same network as SCL:
   #EstadoVI.En_Termico1 := "ON" AND #Termico_Tx;
   #EstadoVI.En_PHS_1 := "ON" AND #pHsMx;
   #EstadoVI.En_pHs_Prot3 := "ON" AND #pHsMx_PR3;
   #EstadoVI.En_Detector_carretilla := "ON" AND #pHsMx_Carretilla;
END_REGION

REGION Network 71: SALIDAS DE LA MESA
   RUNG wire#powerrail
      Contact( "ON" )
      wire#w1
      Contact( "DB1_SalidasExterioresDeMesa".Mesa[#Mesa].Avanzar_E1E3 )
      Contact( #EnMovimiento_Tx )
      Coil( #EstadoVI.Sa_Rod_Avance )
   END_RUNG
   RUNG wire#w1
      Contact( "DB1_SalidasExterioresDeMesa".Mesa[#Mesa].Retroceder_E1E3 )
      Contact( #EnMovimiento_Tx )
      Coil( #EstadoVI.Sa_Rod_Retroc )
   END_RUNG
   // the same network as SCL:
   #EstadoVI.Sa_Rod_Avance := "ON" AND "DB1_SalidasExterioresDeMesa".Mesa[#Mesa].Avanzar_E1E3 AND #EnMovimiento_Tx;
   #EstadoVI.Sa_Rod_Retroc := "ON" AND "DB1_SalidasExterioresDeMesa".Mesa[#Mesa].Retroceder_E1E3 AND #EnMovimiento_Tx;
END_REGION

REGION Network 72: FINALIZAR - Guardar las Variables de Trabajo de la Mesa
   RUNG wire#powerrail
      Move(in := #EstadoVI, out1 => "DB900_Estado_Mesas".EstadoVI[#Mesa])
   END_RUNG
   // the same network as SCL:
   "DB900_Estado_Mesas".EstadoVI[#Mesa] := #EstadoVI;
END_REGION
END_FUNCTION_BLOCK
